LIN {X 0,Y 485.175,Z 367.436,A -85,B 0,C 180,E1 -14967.515,E2 -14967.515} C_VEL
LIN {X 0,Y 481.422,Z 350.009,A -85,B 0,C 180,E1 -14969.767,E2 -14969.767} C_VEL
LIN {X 0,Y 478.767,Z 338.408,A -85,B 0,C 180,E1 -14971.29,E2 -14971.29} C_VEL
LIN {X 0,Y 478.759,Z 338.404,A -85,B 0,C 180,E1 -14973.777,E2 -14973.777} C_VEL
LIN {X 0,Y 478.742,Z 338.407,A -85,B 0,C 180,E1 -14976.861,E2 -14976.861} C_VEL
LIN {X 0,Y 478.759,Z 338.402,A -85,B 0,C 180,E1 -14980.072,E2 -14980.072} C_VEL
LIN {X 0,Y 478.752,Z 338.406,A -85,B 0,C 180,E1 -14983.444,E2 -14983.444} C_VEL
LIN {X 0,Y 478.752,Z 338.406,A -85,B 0,C 180,E1 -14986.556,E2 -14986.556} C_VEL
LIN {X 0,Y 478.766,Z 338.401,A -85,B 0,C 180,E1 -14989.93,E2 -14989.93} C_VEL
LIN {X 0,Y 478.755,Z 338.403,A -85,B 0,C 180,E1 -14993.58,E2 -14993.58} C_VEL
LIN {X 0,Y 478.758,Z 338.409,A -85,B 0,C 180,E1 -14996.506,E2 -14996.506} C_VEL
LIN {X 0,Y 478.73,Z 338.406,A -85,B 0,C 180,E1 -14999.684,E2 -14999.684} C_VEL
LIN {X 0,Y 478.774,Z 338.404,A -85,B 0,C 180,E1 -15002.085,E2 -15002.085} C_VEL
LIN {X 0,Y 478.749,Z 338.404,A -85,B 0,C 180,E1 -15005.109,E2 -15005.109} C_VEL
LIN {X 0,Y 478.778,Z 338.404,A -85,B 0,C 180,E1 -15008.547,E2 -15008.547} C_VEL
LIN {X 0,Y 478.822,Z 338.4,A -85,B 0,C 180,E1 -15011.964,E2 -15011.964} C_VEL
LIN {X 0,Y 478.833,Z 338.4,A -85,B 0,C 180,E1 -15015.708,E2 -15015.708} C_VEL
LIN {X 0,Y 486.096,Z 358.59,A -85,B 0,C 180,E1 -15016.306,E2 -15016.306} C_VEL
LIN {X 0,Y 485.152,Z 454.452,A -85,B 0,C 180,E1 -15017.731,E2 -15017.731} C_VEL
LIN {X 0,Y 485.026,Z 469.135,A -85,B 0,C 180,E1 -15018.072,E2 -15018.072} C_VEL
LIN {X 0,Y 484.751,Z 482.42,A -85,B 0,C 180,E1 -15018.54,E2 -15018.54} C_VEL
LIN {X 0,Y 484.218,Z 495.503,A -85,B 0,C 180,E1 -15019.161,E2 -15019.161} C_VEL
LIN {X 0,Y 483.576,Z 508.953,A -85,B 0,C 180,E1 -15019.99,E2 -15019.99} C_VEL
LIN {X 0,Y 482.964,Z 520.946,A -85,B 0,C 180,E1 -15020.925,E2 -15020.925} C_VEL
LIN {X 0,Y 482.227,Z 530.859,A -85,B 0,C 180,E1 -15021.858,E2 -15021.858} C_VEL
LIN {X 0,Y 481.457,Z 540.12,A -85,B 0,C 180,E1 -15022.897,E2 -15022.897} C_VEL
LIN {X 0,Y 480.63,Z 549.438,A -85,B 0,C 180,E1 -15024.145,E2 -15024.145} C_VEL
LIN {X 0,Y 480.029,Z 557.328,A -85,B 0,C 180,E1 -15025.429,E2 -15025.429} C_VEL
LIN {X 0,Y 479.027,Z 560.589,A -85,B 0,C 180,E1 -15026.007,E2 -15026.007} C_VEL
LIN {X 0,Y 475.742,Z 565.626,A -85,B 0,C 180,E1 -15026.954,E2 -15026.954} C_VEL
LIN {X 0,Y 472.545,Z 570.095,A -85,B 0,C 180,E1 -15027.951,E2 -15027.951} C_VEL
LIN {X 0,Y 471.694,Z 572.465,A -85,B 0,C 180,E1 -15028.599,E2 -15028.599} C_VEL
LIN {X 0,Y 471.381,Z 576.642,A -85,B 0,C 180,E1 -15030,E2 -15030} C_VEL
LIN {X 0,Y 471.202,Z 580.325,A -85,B 0,C 180,E1 -15031.704,E2 -15031.704} C_VEL
LIN {X 0,Y 471.107,Z 582.654,A -85,B 0,C 180,E1 -15033.41,E2 -15033.41} C_VEL
LIN {X 0,Y 471.112,Z 583.684,A -85,B 0,C 180,E1 -15035.118,E2 -15035.118} C_VEL
LIN {X 0,Y 471.242,Z 583.424,A -85,B 0,C 180,E1 -15036.829,E2 -15036.829} C_VEL
LIN {X 0,Y 471.499,Z 581.866,A -85,B 0,C 180,E1 -15038.543,E2 -15038.543} C_VEL
LIN {X 0,Y 471.86,Z 578.968,A -85,B 0,C 180,E1 -15040.261,E2 -15040.261} C_VEL
LIN {X 0,Y 472.534,Z 574.619,A -85,B 0,C 180,E1 -15041.977,E2 -15041.977} C_VEL
LIN {X 0,Y 473.094,Z 570.29,A -85,B 0,C 180,E1 -15043.267,E2 -15043.267} C_VEL
LIN {X 0,Y 473.782,Z 564.997,A -85,B 0,C 180,E1 -15044.556,E2 -15044.556} C_VEL
LIN {X 0,Y 474.765,Z 557.377,A -85,B 0,C 180,E1 -15046.059,E2 -15046.059} C_VEL
LIN {X 0,Y 475.683,Z 549.394,A -85,B 0,C 180,E1 -15047.349,E2 -15047.349} C_VEL
LIN {X 0,Y 476.762,Z 539.731,A -85,B 0,C 180,E1 -15048.636,E2 -15048.636} C_VEL
LIN {X 0,Y 477.733,Z 530.02,A -85,B 0,C 180,E1 -15049.708,E2 -15049.708} C_VEL
LIN {X 0,Y 478.639,Z 519.536,A -85,B 0,C 180,E1 -15050.674,E2 -15050.674} C_VEL
LIN {X 0,Y 479.678,Z 506.651,A -85,B 0,C 180,E1 -15051.636,E2 -15051.636} C_VEL
LIN {X 0,Y 480.39,Z 493.952,A -85,B 0,C 180,E1 -15052.391,E2 -15052.391} C_VEL
LIN {X 0,Y 480.884,Z 480.962,A -85,B 0,C 180,E1 -15052.989,E2 -15052.989} C_VEL
LIN {X 0,Y 481.254,Z 467.044,A -85,B 0,C 180,E1 -15053.452,E2 -15053.452} C_VEL
LIN {X 0,Y 481.406,Z 452.358,A -85,B 0,C 180,E1 -15053.757,E2 -15053.757} C_VEL
LIN {X 0,Y 482.688,Z 365.012,A -85,B 0,C 180,E1 -15055.071,E2 -15055.071} C_VEL
LIN {X 0,Y 472.549,Z 341.866,A -85,B 0,C 180,E1 -15055.964,E2 -15055.964} C_VEL
LIN {X 0,Y 471.684,Z 339.29,A -85,B 0,C 180,E1 -15056.066,E2 -15056.066} C_VEL
LIN {X 0,Y 471.685,Z 339.289,A -85,B 0,C 180,E1 -15059.344,E2 -15059.344} C_VEL
LIN {X 0,Y 471.624,Z 339.297,A -85,B 0,C 180,E1 -15062.321,E2 -15062.321} C_VEL
LIN {X 0,Y 471.636,Z 339.292,A -85,B 0,C 180,E1 -15065.395,E2 -15065.395} C_VEL
LIN {X 0,Y 471.628,Z 339.296,A -85,B 0,C 180,E1 -15068.592,E2 -15068.592} C_VEL
LIN {X 0,Y 471.672,Z 339.29,A -85,B 0,C 180,E1 -15070.8,E2 -15070.8} C_VEL
LIN {X 0,Y 471.685,Z 339.287,A -85,B 0,C 180,E1 -15074.263,E2 -15074.263} C_VEL
LIN {X 0,Y 471.681,Z 339.286,A -85,B 0,C 180,E1 -15076.913,E2 -15076.913} C_VEL
LIN {X 0,Y 471.673,Z 339.286,A -85,B 0,C 180,E1 -15079.233,E2 -15079.233} C_VEL
LIN {X 0,Y 471.624,Z 339.268,A -85,B 0,C 180,E1 -15082.488,E2 -15082.488} C_VEL
LIN {X 0,Y 471.659,Z 339.279,A -85,B 0,C 180,E1 -15085.644,E2 -15085.644} C_VEL
LIN {X 0,Y 471.649,Z 339.282,A -85,B 0,C 180,E1 -15088.682,E2 -15088.682} C_VEL
LIN {X 0,Y 471.696,Z 339.286,A -85,B 0,C 180,E1 -15091.628,E2 -15091.628} C_VEL
LIN {X 0,Y 471.698,Z 339.277,A -85,B 0,C 180,E1 -15094.934,E2 -15094.934} C_VEL
LIN {X 0,Y 471.653,Z 339.283,A -85,B 0,C 180,E1 -15098.206,E2 -15098.206} C_VEL
LIN {X 0,Y 471.723,Z 339.286,A -85,B 0,C 180,E1 -15100.414,E2 -15100.414} C_VEL
LIN {X 0,Y 477.254,Z 358.133,A -85,B 0,C 180,E1 -15100.948,E2 -15100.948} C_VEL
LIN {X 0,Y 475.404,Z 458.142,A -85,B 0,C 180,E1 -15102.884,E2 -15102.884} C_VEL
LIN {X 0,Y 475.207,Z 473.733,A -85,B 0,C 180,E1 -15103.372,E2 -15103.372} C_VEL
LIN {X 0,Y 474.822,Z 488.087,A -85,B 0,C 180,E1 -15103.998,E2 -15103.998} C_VEL
LIN {X 0,Y 474.305,Z 502.141,A -85,B 0,C 180,E1 -15104.803,E2 -15104.803} C_VEL
LIN {X 0,Y 473.779,Z 515.566,A -85,B 0,C 180,E1 -15105.771,E2 -15105.771} C_VEL
LIN {X 0,Y 473.158,Z 527.661,A -85,B 0,C 180,E1 -15106.844,E2 -15106.844} C_VEL
LIN {X 0,Y 472.756,Z 538.588,A -85,B 0,C 180,E1 -15108.028,E2 -15108.028} C_VEL
LIN {X 0,Y 472.269,Z 548.47,A -85,B 0,C 180,E1 -15109.316,E2 -15109.316} C_VEL
LIN {X 0,Y 471.798,Z 556.687,A -85,B 0,C 180,E1 -15110.601,E2 -15110.601} C_VEL
LIN {X 0,Y 471.436,Z 564.576,A -85,B 0,C 180,E1 -15112.1,E2 -15112.1} C_VEL
LIN {X 0,Y 471.186,Z 570.862,A -85,B 0,C 180,E1 -15113.598,E2 -15113.598} C_VEL
LIN {X 0,Y 471.065,Z 575.618,A -85,B 0,C 180,E1 -15115.04,E2 -15115.04} C_VEL
LIN {X 0,Y 471.062,Z 579.426,A -85,B 0,C 180,E1 -15116.59,E2 -15116.59} C_VEL
LIN {X 0,Y 471.048,Z 582.191,A -85,B 0,C 180,E1 -15118.296,E2 -15118.296} C_VEL
LIN {X 0,Y 471.138,Z 583.53,A -85,B 0,C 180,E1 -15120,E2 -15120} C_VEL
LIN {X 0,Y 471.354,Z 583.455,A -85,B 0,C 180,E1 -15121.703,E2 -15121.703} C_VEL
LIN {X 0,Y 471.885,Z 581.884,A -85,B 0,C 180,E1 -15123.404,E2 -15123.404} C_VEL
LIN {X 0,Y 472.565,Z 578.84,A -85,B 0,C 180,E1 -15125.102,E2 -15125.102} C_VEL
LIN {X 0,Y 473.152,Z 574.316,A -85,B 0,C 180,E1 -15126.801,E2 -15126.801} C_VEL
LIN {X 0,Y 474.083,Z 569.426,A -85,B 0,C 180,E1 -15128.145,E2 -15128.145} C_VEL
LIN {X 0,Y 475.187,Z 562.024,A -85,B 0,C 180,E1 -15129.759,E2 -15129.759} C_VEL
LIN {X 0,Y 476.091,Z 554.81,A -85,B 0,C 180,E1 -15131.026,E2 -15131.026} C_VEL
LIN {X 0,Y 477.182,Z 546.051,A -85,B 0,C 180,E1 -15132.289,E2 -15132.289} C_VEL
LIN {X 0,Y 478.244,Z 535.494,A -85,B 0,C 180,E1 -15133.552,E2 -15133.552} C_VEL
LIN {X 0,Y 479.504,Z 523.618,A -85,B 0,C 180,E1 -15134.703,E2 -15134.703} C_VEL
LIN {X 0,Y 480.668,Z 511.003,A -85,B 0,C 180,E1 -15135.681,E2 -15135.681} C_VEL
LIN {X 0,Y 481.659,Z 497.123,A -85,B 0,C 180,E1 -15136.55,E2 -15136.55} C_VEL
LIN {X 0,Y 482.27,Z 483.595,A -85,B 0,C 180,E1 -15137.213,E2 -15137.213} C_VEL
LIN {X 0,Y 482.778,Z 468.86,A -85,B 0,C 180,E1 -15137.739,E2 -15137.739} C_VEL
LIN {X 0,Y 483.214,Z 450.578,A -85,B 0,C 180,E1 -15138.186,E2 -15138.186} C_VEL
LIN {X 0,Y 486.455,Z 378.243,A -85,B 0,C 180,E1 -15139.782,E2 -15139.782} C_VEL
LIN {X 0,Y 486.873,Z 368.471,A -85,B 0,C 180,E1 -15140.011,E2 -15140.011} C_VEL
LIN {X 0,Y 480.186,Z 354.884,A -85,B 0,C 180,E1 -15140.946,E2 -15140.946} C_VEL
LIN {X 0,Y 475.319,Z 346.362,A -85,B 0,C 180,E1 -15141.636,E2 -15141.636} C_VEL
LIN {X 0,Y 473.366,Z 343.01,A -85,B 0,C 180,E1 -15141.922,E2 -15141.922} C_VEL
LIN {X 0,Y 471.939,Z 340.35,A -85,B 0,C 180,E1 -15142.149,E2 -15142.149} C_VEL
LIN {X 0,Y 471.737,Z 339.286,A -85,B 0,C 180,E1 -15142.215,E2 -15142.215} C_VEL
LIN {X 0,Y 471.713,Z 339.288,A -85,B 0,C 180,E1 -15145.507,E2 -15145.507} C_VEL
LIN {X 0,Y 471.71,Z 339.286,A -85,B 0,C 180,E1 -15148.37,E2 -15148.37} C_VEL
LIN {X 0,Y 471.69,Z 339.289,A -85,B 0,C 180,E1 -15151.315,E2 -15151.315} C_VEL
LIN {X 0,Y 471.7,Z 339.282,A -85,B 0,C 180,E1 -15154.352,E2 -15154.352} C_VEL
LIN {X 0,Y 471.67,Z 339.284,A -85,B 0,C 180,E1 -15157.507,E2 -15157.507} C_VEL
LIN {X 0,Y 471.682,Z 339.283,A -85,B 0,C 180,E1 -15159.683,E2 -15159.683} C_VEL
LIN {X 0,Y 471.679,Z 339.285,A -85,B 0,C 180,E1 -15163.086,E2 -15163.086} C_VEL
LIN {X 0,Y 471.686,Z 339.283,A -85,B 0,C 180,E1 -15165.738,E2 -15165.738} C_VEL
LIN {X 0,Y 471.67,Z 339.289,A -85,B 0,C 180,E1 -15169.232,E2 -15169.232} C_VEL
LIN {X 0,Y 471.622,Z 339.298,A -85,B 0,C 180,E1 -15172.488,E2 -15172.488} C_VEL
LIN {X 0,Y 471.629,Z 339.285,A -85,B 0,C 180,E1 -15175.642,E2 -15175.642} C_VEL
LIN {X 0,Y 471.674,Z 339.381,A -85,B 0,C 180,E1 -15177.525,E2 -15177.525} C_VEL
LIN {X 0,Y 475.594,Z 355.323,A -85,B 0,C 180,E1 -15180.107,E2 -15180.107} C_VEL
LIN {X 0,Y 478.251,Z 367.913,A -85,B 0,C 180,E1 -15182.052,E2 -15182.052} C_VEL
LIN {X 0,Y 478.074,Z 372.934,A -85,B 0,C 180,E1 -15182.751,E2 -15182.751} C_VEL
LIN {X 0,Y 475.774,Z 399.746,A -85,B 0,C 180,E1 -15186.378,E2 -15186.378} C_VEL
LIN {X 0,Y 475.192,Z 407.187,A -85,B 0,C 180,E1 -15187.379,E2 -15187.379} C_VEL
LIN {X 0,Y 478.527,Z 428.614,A -85,B 0,C 180,E1 -15188.267,E2 -15188.267} C_VEL
LIN {X 0,Y 480.639,Z 445.485,A -85,B 0,C 180,E1 -15188.882,E2 -15188.882} C_VEL
LIN {X 0,Y 482.569,Z 472.55,A -85,B 0,C 180,E1 -15189.724,E2 -15189.724} C_VEL
LIN {X 0,Y 480.102,Z 533.094,A -85,B 0,C 180,E1 -15191.03,E2 -15191.03} C_VEL
LIN {X 0,Y 479.615,Z 559.637,A -85,B 0,C 180,E1 -15191.452,E2 -15191.452} C_VEL
LIN {X 0,Y 478.87,Z 573.984,A -85,B 0,C 180,E1 -15191.836,E2 -15191.836} C_VEL
LIN {X 0,Y 477.735,Z 588.728,A -85,B 0,C 180,E1 -15192.415,E2 -15192.415} C_VEL
LIN {X 0,Y 476.54,Z 602.089,A -85,B 0,C 180,E1 -15193.124,E2 -15193.124} C_VEL
LIN {X 0,Y 475.343,Z 614.425,A -85,B 0,C 180,E1 -15193.961,E2 -15193.961} C_VEL
LIN {X 0,Y 474.022,Z 626.919,A -85,B 0,C 180,E1 -15195.013,E2 -15195.013} C_VEL
LIN {X 0,Y 472.917,Z 637.198,A -85,B 0,C 180,E1 -15196.073,E2 -15196.073} C_VEL
LIN {X 0,Y 472.057,Z 647.255,A -85,B 0,C 180,E1 -15197.303,E2 -15197.303} C_VEL
LIN {X 0,Y 471.418,Z 658.908,A -85,B 0,C 180,E1 -15198.472,E2 -15198.472} C_VEL
LIN {X 0,Y 470.946,Z 669.094,A -85,B 0,C 180,E1 -15199.719,E2 -15199.719} C_VEL
LIN {X 0,Y 470.512,Z 677.788,A -85,B 0,C 180,E1 -15201.007,E2 -15201.007} C_VEL
LIN {X 0,Y 470.174,Z 686.056,A -85,B 0,C 180,E1 -15202.51,E2 -15202.51} C_VEL
LIN {X 0,Y 470.009,Z 692.665,A -85,B 0,C 180,E1 -15204.012,E2 -15204.012} C_VEL
LIN {X 0,Y 469.925,Z 697.153,A -85,B 0,C 180,E1 -15205.297,E2 -15205.297} C_VEL
LIN {X 0,Y 469.843,Z 700.68,A -85,B 0,C 180,E1 -15206.581,E2 -15206.581} C_VEL
LIN {X 0,Y 469.856,Z 702.494,A -85,B 0,C 180,E1 -15207.437,E2 -15207.437} C_VEL
LIN {X 0,Y 469.847,Z 704.973,A -85,B 0,C 180,E1 -15209.146,E2 -15209.146} C_VEL
LIN {X 0,Y 469.83,Z 705.968,A -85,B 0,C 180,E1 -15210.854,E2 -15210.854} C_VEL
LIN {X 0,Y 469.856,Z 705.494,A -85,B 0,C 180,E1 -15212.563,E2 -15212.563} C_VEL
LIN {X 0,Y 469.942,Z 703.555,A -85,B 0,C 180,E1 -15214.274,E2 -15214.274} C_VEL
LIN {X 0,Y 470.23,Z 700.082,A -85,B 0,C 180,E1 -15215.985,E2 -15215.985} C_VEL
LIN {X 0,Y 470.588,Z 695.019,A -85,B 0,C 180,E1 -15217.698,E2 -15217.698} C_VEL
LIN {X 0,Y 471.087,Z 690.095,A -85,B 0,C 180,E1 -15218.982,E2 -15218.982} C_VEL
LIN {X 0,Y 471.897,Z 682.967,A -85,B 0,C 180,E1 -15220.476,E2 -15220.476} C_VEL
LIN {X 0,Y 472.829,Z 674.129,A -85,B 0,C 180,E1 -15221.97,E2 -15221.97} C_VEL
LIN {X 0,Y 473.827,Z 664.913,A -85,B 0,C 180,E1 -15223.246,E2 -15223.246} C_VEL
LIN {X 0,Y 475.122,Z 653.768,A -85,B 0,C 180,E1 -15224.514,E2 -15224.514} C_VEL
LIN {X 0,Y 476.226,Z 642.496,A -85,B 0,C 180,E1 -15225.571,E2 -15225.571} C_VEL
LIN {X 0,Y 477.639,Z 628.699,A -85,B 0,C 180,E1 -15226.616,E2 -15226.616} C_VEL
LIN {X 0,Y 478.836,Z 614.862,A -85,B 0,C 180,E1 -15227.45,E2 -15227.45} C_VEL
LIN {X 0,Y 479.94,Z 600.174,A -85,B 0,C 180,E1 -15228.121,E2 -15228.121} C_VEL
LIN {X 0,Y 480.96,Z 584.717,A -85,B 0,C 180,E1 -15228.631,E2 -15228.631} C_VEL
LIN {X 0,Y 485.642,Z 483.73,A -85,B 0,C 180,E1 -15230.914,E2 -15230.914} C_VEL
LIN {X 0,Y 486.051,Z 471.893,A -85,B 0,C 180,E1 -15231.207,E2 -15231.207} C_VEL
LIN {X 0,Y 485.065,Z 454.594,A -85,B 0,C 180,E1 -15231.77,E2 -15231.77} C_VEL
LIN {X 0,Y 482.938,Z 436.376,A -85,B 0,C 180,E1 -15232.478,E2 -15232.478} C_VEL
LIN {X 0,Y 481.981,Z 418.453,A -85,B 0,C 180,E1 -15233.573,E2 -15233.573} C_VEL
LIN {X 0,Y 480.737,Z 398.185,A -85,B 0,C 180,E1 -15234.995,E2 -15234.995} C_VEL
LIN {X 0,Y 479.656,Z 383.288,A -85,B 0,C 180,E1 -15236.196,E2 -15236.196} C_VEL
LIN {X 0,Y 479.315,Z 374.608,A -85,B 0,C 180,E1 -15236.948,E2 -15236.948} C_VEL
LIN {X 0,Y 478.81,Z 365.879,A -85,B 0,C 180,E1 -15237.783,E2 -15237.783} C_VEL
LIN {X 0,Y 476.954,Z 356.575,A -85,B 0,C 180,E1 -15238.988,E2 -15238.988} C_VEL
LIN {X 0,Y 474.733,Z 345.236,A -85,B 0,C 180,E1 -15240.717,E2 -15240.717} C_VEL
LIN {X 0,Y 474.115,Z 343.792,A -85,B 0,C 180,E1 -15241.032,E2 -15241.032} C_VEL
LIN {X 0,Y 472.071,Z 340.988,A -85,B 0,C 180,E1 -15241.91,E2 -15241.91} C_VEL
LIN {X 0,Y 471.613,Z 339.294,A -85,B 0,C 180,E1 -15242.322,E2 -15242.322} C_VEL
LIN {X 0,Y 471.624,Z 339.292,A -85,B 0,C 180,E1 -15245.396,E2 -15245.396} C_VEL
LIN {X 0,Y 471.622,Z 339.295,A -85,B 0,C 180,E1 -15248.592,E2 -15248.592} C_VEL
LIN {X 0,Y 471.667,Z 339.288,A -85,B 0,C 180,E1 -15250.8,E2 -15250.8} C_VEL
LIN {X 0,Y 471.681,Z 339.291,A -85,B 0,C 180,E1 -15254.263,E2 -15254.263} C_VEL
LIN {X 0,Y 471.664,Z 339.287,A -85,B 0,C 180,E1 -15256.912,E2 -15256.912} C_VEL
LIN {X 0,Y 471.668,Z 339.29,A -85,B 0,C 180,E1 -15259.233,E2 -15259.233} C_VEL
LIN {X 0,Y 471.648,Z 339.291,A -85,B 0,C 180,E1 -15260.47,E2 -15260.47} C_VEL
LIN {X 0,Y 472.464,Z 341.824,A -85,B 0,C 180,E1 -15261.214,E2 -15261.214} C_VEL
LIN {X 0,Y 474.12,Z 344.845,A -85,B 0,C 180,E1 -15262.195,E2 -15262.195} C_VEL
LIN {X 0,Y 477.879,Z 353.112,A -85,B 0,C 180,E1 -15264.437,E2 -15264.437} C_VEL
LIN {X 0,Y 481.184,Z 361.878,A -85,B 0,C 180,E1 -15266.416,E2 -15266.416} C_VEL
LIN {X 0,Y 483.952,Z 370.881,A -85,B 0,C 180,E1 -15268.196,E2 -15268.196} C_VEL
LIN {X 0,Y 486.231,Z 379.99,A -85,B 0,C 180,E1 -15269.807,E2 -15269.807} C_VEL
LIN {X 0,Y 486.938,Z 383.965,A -85,B 0,C 180,E1 -15270.459,E2 -15270.459} C_VEL
LIN {X 0,Y 486.785,Z 387.543,A -85,B 0,C 180,E1 -15270.946,E2 -15270.946} C_VEL
LIN {X 0,Y 484.134,Z 412.267,A -85,B 0,C 180,E1 -15274.03,E2 -15274.03} C_VEL
LIN {X 0,Y 481.588,Z 440.052,A -85,B 0,C 180,E1 -15277.429,E2 -15277.429} C_VEL
LIN {X 0,Y 485.077,Z 458.784,A -85,B 0,C 180,E1 -15278.258,E2 -15278.258} C_VEL
LIN {X 0,Y 486.657,Z 471.979,A -85,B 0,C 180,E1 -15278.747,E2 -15278.747} C_VEL
LIN {X 0,Y 482.69,Z 556.46,A -85,B 0,C 180,E1 -15280.645,E2 -15280.645} C_VEL
LIN {X 0,Y 481.474,Z 583.391,A -85,B 0,C 180,E1 -15281.26,E2 -15281.26} C_VEL
LIN {X 0,Y 480.568,Z 596.124,A -85,B 0,C 180,E1 -15281.683,E2 -15281.683} C_VEL
LIN {X 0,Y 479.389,Z 610.913,A -85,B 0,C 180,E1 -15282.351,E2 -15282.351} C_VEL
LIN {X 0,Y 478.219,Z 624.997,A -85,B 0,C 180,E1 -15283.185,E2 -15283.185} C_VEL
LIN {X 0,Y 476.917,Z 637.696,A -85,B 0,C 180,E1 -15284.125,E2 -15284.125} C_VEL
LIN {X 0,Y 475.637,Z 649.296,A -85,B 0,C 180,E1 -15285.175,E2 -15285.175} C_VEL
LIN {X 0,Y 474.467,Z 659.905,A -85,B 0,C 180,E1 -15286.338,E2 -15286.338} C_VEL
LIN {X 0,Y 473.279,Z 669.716,A -85,B 0,C 180,E1 -15287.631,E2 -15287.631} C_VEL
LIN {X 0,Y 472.382,Z 678.846,A -85,B 0,C 180,E1 -15289.102,E2 -15289.102} C_VEL
LIN {X 0,Y 471.36,Z 686.341,A -85,B 0,C 180,E1 -15290.592,E2 -15290.592} C_VEL
LIN {X 0,Y 470.839,Z 691.557,A -85,B 0,C 180,E1 -15291.876,E2 -15291.876} C_VEL
LIN {X 0,Y 470.435,Z 695.757,A -85,B 0,C 180,E1 -15293.159,E2 -15293.159} C_VEL
LIN {X 0,Y 470.034,Z 699.981,A -85,B 0,C 180,E1 -15294.87,E2 -15294.87} C_VEL
LIN {X 0,Y 469.847,Z 702.671,A -85,B 0,C 180,E1 -15296.582,E2 -15296.582} C_VEL
LIN {X 0,Y 469.765,Z 703.876,A -85,B 0,C 180,E1 -15298.291,E2 -15298.291} C_VEL
LIN {X 0,Y 469.76,Z 703.636,A -85,B 0,C 180,E1 -15300,E2 -15300} C_VEL
LIN {X 0,Y 469.76,Z 701.944,A -85,B 0,C 180,E1 -15301.709,E2 -15301.709} C_VEL
LIN {X 0,Y 469.809,Z 698.766,A -85,B 0,C 180,E1 -15303.419,E2 -15303.419} C_VEL
LIN {X 0,Y 469.863,Z 695.314,A -85,B 0,C 180,E1 -15304.703,E2 -15304.703} C_VEL
LIN {X 0,Y 469.993,Z 690.848,A -85,B 0,C 180,E1 -15306.008,E2 -15306.008} C_VEL
LIN {X 0,Y 470.256,Z 684.46,A -85,B 0,C 180,E1 -15307.489,E2 -15307.489} C_VEL
LIN {X 0,Y 470.579,Z 676.37,A -85,B 0,C 180,E1 -15308.992,E2 -15308.992} C_VEL
LIN {X 0,Y 471.047,Z 667.898,A -85,B 0,C 180,E1 -15310.279,E2 -15310.279} C_VEL
LIN {X 0,Y 471.568,Z 658.05,A -85,B 0,C 180,E1 -15311.524,E2 -15311.524} C_VEL
LIN {X 0,Y 472.122,Z 647.404,A -85,B 0,C 180,E1 -15312.641,E2 -15312.641} C_VEL
LIN {X 0,Y 472.792,Z 634.963,A -85,B 0,C 180,E1 -15313.712,E2 -15313.712} C_VEL
LIN {X 0,Y 473.52,Z 622.844,A -85,B 0,C 180,E1 -15314.565,E2 -15314.565} C_VEL
LIN {X 0,Y 474.22,Z 608.634,A -85,B 0,C 180,E1 -15315.364,E2 -15315.364} C_VEL
LIN {X 0,Y 474.712,Z 594.201,A -85,B 0,C 180,E1 -15315.979,E2 -15315.979} C_VEL
LIN {X 0,Y 475.181,Z 579.664,A -85,B 0,C 180,E1 -15316.417,E2 -15316.417} C_VEL
LIN {X 0,Y 477.528,Z 466.879,A -85,B 0,C 180,E1 -15318.632,E2 -15318.632} C_VEL
LIN {X 0,Y 474.708,Z 439.522,A -85,B 0,C 180,E1 -15319.275,E2 -15319.275} C_VEL
LIN {X 0,Y 476.23,Z 408.418,A -85,B 0,C 180,E1 -15322.94,E2 -15322.94} C_VEL
LIN {X 0,Y 477.57,Z 383.579,A -85,B 0,C 180,E1 -15325.871,E2 -15325.871} C_VEL
LIN {X 0,Y 478.296,Z 370.046,A -85,B 0,C 180,E1 -15327.472,E2 -15327.472} C_VEL
LIN {X 0,Y 477.248,Z 363.687,A -85,B 0,C 180,E1 -15328.285,E2 -15328.285} C_VEL
LIN {X 0,Y 472.51,Z 342.754,A -85,B 0,C 180,E1 -15331.04,E2 -15331.04} C_VEL
LIN {X 0,Y 471.716,Z 339.286,A -85,B 0,C 180,E1 -15331.5,E2 -15331.5} C_VEL
LIN {X 0,Y 471.701,Z 339.281,A -85,B 0,C 180,E1 -15334.352,E2 -15334.352} C_VEL
LIN {X 0,Y 471.671,Z 339.289,A -85,B 0,C 180,E1 -15337.508,E2 -15337.508} C_VEL
LIN {X 0,Y 471.721,Z 339.28,A -85,B 0,C 180,E1 -15339.68,E2 -15339.68} C_VEL
LIN {X 0,Y 471.697,Z 339.286,A -85,B 0,C 180,E1 -15343.312,E2 -15343.312} C_VEL
LIN {X 0,Y 471.707,Z 339.281,A -85,B 0,C 180,E1 -15345.74,E2 -15345.74} C_VEL
LIN {X 0,Y 471.707,Z 339.284,A -85,B 0,C 180,E1 -15349.228,E2 -15349.228} C_VEL
LIN {X 0,Y 471.663,Z 339.286,A -85,B 0,C 180,E1 -15351.914,E2 -15351.914} C_VEL
LIN {X 0,Y 471.699,Z 339.288,A -85,B 0,C 180,E1 -15354.758,E2 -15354.758} C_VEL
LIN {X 0,Y 471.694,Z 339.283,A -85,B 0,C 180,E1 -15357.826,E2 -15357.826} C_VEL
LIN {X 0,Y 471.69,Z 339.288,A -85,B 0,C 180,E1 -15360.657,E2 -15360.657} C_VEL
LIN {X 0,Y 471.693,Z 339.282,A -85,B 0,C 180,E1 -15363.545,E2 -15363.545} C_VEL
LIN {X 0,Y 471.68,Z 339.291,A -85,B 0,C 180,E1 -15366.362,E2 -15366.362} C_VEL
LIN {X 0,Y 471.758,Z 339.274,A -85,B 0,C 180,E1 -15369.293,E2 -15369.293} C_VEL
LIN {X 0,Y 471.727,Z 339.279,A -85,B 0,C 180,E1 -15372.724,E2 -15372.724} C_VEL
LIN {X 0,Y 471.783,Z 339.31,A -85,B 0,C 180,E1 -15375.451,E2 -15375.451} C_VEL
LIN {X 0,Y 479.432,Z 360.627,A -85,B 0,C 180,E1 -15376.085,E2 -15376.085} C_VEL
LIN {X 0,Y 478.337,Z 454.876,A -85,B 0,C 180,E1 -15377.5,E2 -15377.5} C_VEL
LIN {X 0,Y 478.205,Z 469.692,A -85,B 0,C 180,E1 -15377.845,E2 -15377.845} C_VEL
LIN {X 0,Y 477.936,Z 483.032,A -85,B 0,C 180,E1 -15378.321,E2 -15378.321} C_VEL
LIN {X 0,Y 477.417,Z 495.178,A -85,B 0,C 180,E1 -15378.898,E2 -15378.898} C_VEL
LIN {X 0,Y 476.824,Z 507.302,A -85,B 0,C 180,E1 -15379.633,E2 -15379.633} C_VEL
LIN {X 0,Y 476.228,Z 519.045,A -85,B 0,C 180,E1 -15380.522,E2 -15380.522} C_VEL
LIN {X 0,Y 475.475,Z 529.982,A -85,B 0,C 180,E1 -15381.529,E2 -15381.529} C_VEL
LIN {X 0,Y 474.656,Z 539.52,A -85,B 0,C 180,E1 -15382.581,E2 -15382.581} C_VEL
LIN {X 0,Y 473.743,Z 549.071,A -85,B 0,C 180,E1 -15383.847,E2 -15383.847} C_VEL
LIN {X 0,Y 473.162,Z 556.969,A -85,B 0,C 180,E1 -15385.117,E2 -15385.117} C_VEL
LIN {X 0,Y 472.38,Z 564.575,A -85,B 0,C 180,E1 -15386.6,E2 -15386.6} C_VEL
LIN {X 0,Y 471.964,Z 569.878,A -85,B 0,C 180,E1 -15387.874,E2 -15387.874} C_VEL
LIN {X 0,Y 471.694,Z 572.465,A -85,B 0,C 180,E1 -15388.599,E2 -15388.599} C_VEL
LIN {X 0,Y 470.861,Z 574.662,A -85,B 0,C 180,E1 -15389.26,E2 -15389.26} C_VEL
LIN {X 0,Y 467.796,Z 577.914,A -85,B 0,C 180,E1 -15390.342,E2 -15390.342} C_VEL
LIN {X 0,Y 465.29,Z 580.129,A -85,B 0,C 180,E1 -15391.229,E2 -15391.229} C_VEL
LIN {X 0,Y 464.229,Z 581.485,A -85,B 0,C 180,E1 -15391.927,E2 -15391.927} C_VEL
LIN {X 0,Y 464.148,Z 581.826,A -85,B 0,C 180,E1 -15392.166,E2 -15392.166} C_VEL
LIN {X 0,Y 464.04,Z 583.466,A -85,B 0,C 180,E1 -15393.462,E2 -15393.462} C_VEL
LIN {X 0,Y 464.071,Z 584.46,A -85,B 0,C 180,E1 -15395.196,E2 -15395.196} C_VEL
LIN {X 0,Y 464.215,Z 584.167,A -85,B 0,C 180,E1 -15396.933,E2 -15396.933} C_VEL
LIN {X 0,Y 464.465,Z 582.577,A -85,B 0,C 180,E1 -15398.674,E2 -15398.674} C_VEL
LIN {X 0,Y 464.886,Z 579.64,A -85,B 0,C 180,E1 -15400.417,E2 -15400.417} C_VEL
LIN {X 0,Y 465.586,Z 575.254,A -85,B 0,C 180,E1 -15402.159,E2 -15402.159} C_VEL
LIN {X 0,Y 466.168,Z 570.886,A -85,B 0,C 180,E1 -15403.468,E2 -15403.468} C_VEL
LIN {X 0,Y 466.904,Z 565.549,A -85,B 0,C 180,E1 -15404.776,E2 -15404.776} C_VEL
LIN {X 0,Y 467.925,Z 557.881,A -85,B 0,C 180,E1 -15406.301,E2 -15406.301} C_VEL
LIN {X 0,Y 468.889,Z 549.843,A -85,B 0,C 180,E1 -15407.608,E2 -15407.608} C_VEL
LIN {X 0,Y 470.013,Z 540.115,A -85,B 0,C 180,E1 -15408.913,E2 -15408.913} C_VEL
LIN {X 0,Y 471.035,Z 530.326,A -85,B 0,C 180,E1 -15410,E2 -15410} C_VEL
LIN {X 0,Y 472,Z 519.744,A -85,B 0,C 180,E1 -15410.978,E2 -15410.978} C_VEL
LIN {X 0,Y 472.932,Z 508.31,A -85,B 0,C 180,E1 -15411.847,E2 -15411.847} C_VEL
LIN {X 0,Y 473.715,Z 495.842,A -85,B 0,C 180,E1 -15412.609,E2 -15412.609} C_VEL
LIN {X 0,Y 474.214,Z 483.203,A -85,B 0,C 180,E1 -15413.216,E2 -15413.216} C_VEL
LIN {X 0,Y 474.627,Z 468.884,A -85,B 0,C 180,E1 -15413.716,E2 -15413.716} C_VEL
LIN {X 0,Y 474.805,Z 455.104,A -85,B 0,C 180,E1 -15414.024,E2 -15414.024} C_VEL
LIN {X 0,Y 476.177,Z 366.885,A -85,B 0,C 180,E1 -15415.37,E2 -15415.37} C_VEL
LIN {X 0,Y 465.674,Z 343.092,A -85,B 0,C 180,E1 -15416.315,E2 -15416.315} C_VEL
LIN {X 0,Y 464.624,Z 340.17,A -85,B 0,C 180,E1 -15416.423,E2 -15416.423} C_VEL
LIN {X 0,Y 464.668,Z 340.164,A -85,B 0,C 180,E1 -15419.037,E2 -15419.037} C_VEL
LIN {X 0,Y 464.597,Z 340.172,A -85,B 0,C 180,E1 -15422.405,E2 -15422.405} C_VEL
LIN {X 0,Y 464.583,Z 340.171,A -85,B 0,C 180,E1 -15425.496,E2 -15425.496} C_VEL
LIN {X 0,Y 464.585,Z 340.176,A -85,B 0,C 180,E1 -15428.372,E2 -15428.372} C_VEL
LIN {X 0,Y 464.622,Z 340.169,A -85,B 0,C 180,E1 -15431.554,E2 -15431.554} C_VEL
LIN {X 0,Y 464.671,Z 340.156,A -85,B 0,C 180,E1 -15435.112,E2 -15435.112} C_VEL
LIN {X 0,Y 464.629,Z 340.165,A -85,B 0,C 180,E1 -15438.446,E2 -15438.446} C_VEL
LIN {X 0,Y 464.575,Z 340.155,A -85,B 0,C 180,E1 -15441.818,E2 -15441.818} C_VEL
LIN {X 0,Y 464.621,Z 340.151,A -85,B 0,C 180,E1 -15445.049,E2 -15445.049} C_VEL
LIN {X 0,Y 464.582,Z 340.167,A -85,B 0,C 180,E1 -15448.15,E2 -15448.15} C_VEL
LIN {X 0,Y 464.659,Z 340.158,A -85,B 0,C 180,E1 -15451.159,E2 -15451.159} C_VEL
LIN {X 0,Y 464.648,Z 340.156,A -85,B 0,C 180,E1 -15454.076,E2 -15454.076} C_VEL
LIN {X 0,Y 464.63,Z 340.164,A -85,B 0,C 180,E1 -15456.923,E2 -15456.923} C_VEL
LIN {X 0,Y 464.692,Z 340.163,A -85,B 0,C 180,E1 -15460.243,E2 -15460.243} C_VEL
LIN {X 0,Y 470.238,Z 358.755,A -85,B 0,C 180,E1 -15460.781,E2 -15460.781} C_VEL
LIN {X 0,Y 468.391,Z 458.568,A -85,B 0,C 180,E1 -15462.759,E2 -15462.759} C_VEL
LIN {X 0,Y 468.183,Z 473.722,A -85,B 0,C 180,E1 -15463.237,E2 -15463.237} C_VEL
LIN {X 0,Y 467.817,Z 488.047,A -85,B 0,C 180,E1 -15463.863,E2 -15463.863} C_VEL
LIN {X 0,Y 467.346,Z 500.625,A -85,B 0,C 180,E1 -15464.571,E2 -15464.571} C_VEL
LIN {X 0,Y 466.892,Z 513.081,A -85,B 0,C 180,E1 -15465.446,E2 -15465.446} C_VEL
LIN {X 0,Y 466.269,Z 525.734,A -85,B 0,C 180,E1 -15466.535,E2 -15466.535} C_VEL
LIN {X 0,Y 465.81,Z 536.226,A -85,B 0,C 180,E1 -15467.626,E2 -15467.626} C_VEL
LIN {X 0,Y 465.34,Z 546.718,A -85,B 0,C 180,E1 -15468.935,E2 -15468.935} C_VEL
LIN {X 0,Y 464.871,Z 555.375,A -85,B 0,C 180,E1 -15470.24,E2 -15470.24} C_VEL
LIN {X 0,Y 464.452,Z 563.643,A -85,B 0,C 180,E1 -15471.763,E2 -15471.763} C_VEL
LIN {X 0,Y 464.198,Z 569.45,A -85,B 0,C 180,E1 -15473.066,E2 -15473.066} C_VEL
LIN {X 0,Y 464.031,Z 574.203,A -85,B 0,C 180,E1 -15474.369,E2 -15474.369} C_VEL
LIN {X 0,Y 463.997,Z 577.973,A -85,B 0,C 180,E1 -15475.671,E2 -15475.671} C_VEL
LIN {X 0,Y 464.027,Z 581.62,A -85,B 0,C 180,E1 -15477.404,E2 -15477.404} C_VEL
LIN {X 0,Y 464.023,Z 583.789,A -85,B 0,C 180,E1 -15479.135,E2 -15479.135} C_VEL
LIN {X 0,Y 464.206,Z 584.536,A -85,B 0,C 180,E1 -15480.864,E2 -15480.864} C_VEL
LIN {X 0,Y 464.567,Z 583.856,A -85,B 0,C 180,E1 -15482.592,E2 -15482.592} C_VEL
LIN {X 0,Y 465.247,Z 581.691,A -85,B 0,C 180,E1 -15484.317,E2 -15484.317} C_VEL
LIN {X 0,Y 465.907,Z 578.029,A -85,B 0,C 180,E1 -15486.041,E2 -15486.041} C_VEL
LIN {X 0,Y 466.645,Z 573.765,A -85,B 0,C 180,E1 -15487.476,E2 -15487.476} C_VEL
LIN {X 0,Y 467.781,Z 567.63,A -85,B 0,C 180,E1 -15489.046,E2 -15489.046} C_VEL
LIN {X 0,Y 468.817,Z 560.255,A -85,B 0,C 180,E1 -15490.546,E2 -15490.546} C_VEL
LIN {X 0,Y 469.915,Z 552.488,A -85,B 0,C 180,E1 -15491.827,E2 -15491.827} C_VEL
LIN {X 0,Y 471.066,Z 543.089,A -85,B 0,C 180,E1 -15493.106,E2 -15493.106} C_VEL
LIN {X 0,Y 472.213,Z 532.661,A -85,B 0,C 180,E1 -15494.276,E2 -15494.276} C_VEL
LIN {X 0,Y 473.446,Z 521.174,A -85,B 0,C 180,E1 -15495.334,E2 -15495.334} C_VEL
LIN {X 0,Y 474.636,Z 508.487,A -85,B 0,C 180,E1 -15496.283,E2 -15496.283} C_VEL
LIN {X 0,Y 475.542,Z 494.215,A -85,B 0,C 180,E1 -15497.133,E2 -15497.133} C_VEL
LIN {X 0,Y 476.201,Z 480.339,A -85,B 0,C 180,E1 -15497.771,E2 -15497.771} C_VEL
LIN {X 0,Y 476.633,Z 465.882,A -85,B 0,C 180,E1 -15498.252,E2 -15498.252} C_VEL
LIN {X 0,Y 478.747,Z 412.507,A -85,B 0,C 180,E1 -15499.469,E2 -15499.469} C_VEL
LIN {X 0,Y 480.866,Z 370.711,A -85,B 0,C 180,E1 -15500.44,E2 -15500.44} C_VEL
LIN {X 0,Y 474.525,Z 357.886,A -85,B 0,C 180,E1 -15501.367,E2 -15501.367} C_VEL
LIN {X 0,Y 468.562,Z 347.551,A -85,B 0,C 180,E1 -15502.263,E2 -15502.263} C_VEL
LIN {X 0,Y 466.675,Z 344.252,A -85,B 0,C 180,E1 -15502.564,E2 -15502.564} C_VEL
LIN {X 0,Y 465.07,Z 341.72,A -85,B 0,C 180,E1 -15502.814,E2 -15502.814} C_VEL
LIN {X 0,Y 464.688,Z 340.163,A -85,B 0,C 180,E1 -15502.914,E2 -15502.914} C_VEL
LIN {X 0,Y 464.668,Z 340.165,A -85,B 0,C 180,E1 -15505.922,E2 -15505.922} C_VEL
LIN {X 0,Y 464.674,Z 340.16,A -85,B 0,C 180,E1 -15509.039,E2 -15509.039} C_VEL
LIN {X 0,Y 464.652,Z 340.162,A -85,B 0,C 180,E1 -15512.415,E2 -15512.415} C_VEL
LIN {X 0,Y 464.645,Z 340.159,A -85,B 0,C 180,E1 -15515.507,E2 -15515.507} C_VEL
LIN {X 0,Y 464.615,Z 340.16,A -85,B 0,C 180,E1 -15518.377,E2 -15518.377} C_VEL
LIN {X 0,Y 464.627,Z 340.162,A -85,B 0,C 180,E1 -15521.553,E2 -15521.553} C_VEL
LIN {X 0,Y 464.669,Z 340.159,A -85,B 0,C 180,E1 -15524.888,E2 -15524.888} C_VEL
LIN {X 0,Y 464.632,Z 340.163,A -85,B 0,C 180,E1 -15527.62,E2 -15527.62} C_VEL
LIN {X 0,Y 464.599,Z 340.174,A -85,B 0,C 180,E1 -15530.713,E2 -15530.713} C_VEL
LIN {X 0,Y 464.564,Z 340.175,A -85,B 0,C 180,E1 -15533.983,E2 -15533.983} C_VEL
LIN {X 0,Y 464.623,Z 340.253,A -85,B 0,C 180,E1 -15537.193,E2 -15537.193} C_VEL
LIN {X 0,Y 468.583,Z 356.222,A -85,B 0,C 180,E1 -15539.829,E2 -15539.829} C_VEL
LIN {X 0,Y 471.311,Z 369.013,A -85,B 0,C 180,E1 -15541.845,E2 -15541.845} C_VEL
LIN {X 0,Y 471.367,Z 372.377,A -85,B 0,C 180,E1 -15542.33,E2 -15542.33} C_VEL
LIN {X 0,Y 469.231,Z 396.044,A -85,B 0,C 180,E1 -15545.585,E2 -15545.585} C_VEL
LIN {X 0,Y 468.554,Z 404.474,A -85,B 0,C 180,E1 -15546.735,E2 -15546.735} C_VEL
LIN {X 0,Y 472.4,Z 428.96,A -85,B 0,C 180,E1 -15547.784,E2 -15547.784} C_VEL
LIN {X 0,Y 474.525,Z 445.801,A -85,B 0,C 180,E1 -15548.425,E2 -15548.425} C_VEL
LIN {X 0,Y 476.415,Z 473.278,A -85,B 0,C 180,E1 -15549.313,E2 -15549.313} C_VEL
LIN {X 0,Y 473.203,Z 546.714,A -85,B 0,C 180,E1 -15550.939,E2 -15550.939} C_VEL
LIN {X 0,Y 472.808,Z 563.547,A -85,B 0,C 180,E1 -15551.259,E2 -15551.259} C_VEL
LIN {X 0,Y 471.946,Z 577.093,A -85,B 0,C 180,E1 -15551.672,E2 -15551.672} C_VEL
LIN {X 0,Y 470.755,Z 591.103,A -85,B 0,C 180,E1 -15552.274,E2 -15552.274} C_VEL
LIN {X 0,Y 469.582,Z 603.511,A -85,B 0,C 180,E1 -15552.978,E2 -15552.978} C_VEL
LIN {X 0,Y 468.377,Z 615.416,A -85,B 0,C 180,E1 -15553.827,E2 -15553.827} C_VEL
LIN {X 0,Y 467.016,Z 627.518,A -85,B 0,C 180,E1 -15554.894,E2 -15554.894} C_VEL
LIN {X 0,Y 465.775,Z 638.474,A -85,B 0,C 180,E1 -15556.077,E2 -15556.077} C_VEL
LIN {X 0,Y 464.91,Z 648.197,A -85,B 0,C 180,E1 -15557.326,E2 -15557.326} C_VEL
LIN {X 0,Y 464.332,Z 659.306,A -85,B 0,C 180,E1 -15558.47,E2 -15558.47} C_VEL
LIN {X 0,Y 463.819,Z 669.713,A -85,B 0,C 180,E1 -15559.779,E2 -15559.779} C_VEL
LIN {X 0,Y 463.394,Z 678.313,A -85,B 0,C 180,E1 -15561.087,E2 -15561.087} C_VEL
LIN {X 0,Y 463.087,Z 686.498,A -85,B 0,C 180,E1 -15562.613,E2 -15562.613} C_VEL
LIN {X 0,Y 462.931,Z 692.17,A -85,B 0,C 180,E1 -15563.92,E2 -15563.92} C_VEL
LIN {X 0,Y 462.845,Z 696.769,A -85,B 0,C 180,E1 -15565.225,E2 -15565.225} C_VEL
LIN {X 0,Y 462.751,Z 700.378,A -85,B 0,C 180,E1 -15566.529,E2 -15566.529} C_VEL
LIN {X 0,Y 462.77,Z 702.261,A -85,B 0,C 180,E1 -15567.397,E2 -15567.397} C_VEL
LIN {X 0,Y 462.755,Z 704.837,A -85,B 0,C 180,E1 -15569.133,E2 -15569.133} C_VEL
LIN {X 0,Y 462.739,Z 705.927,A -85,B 0,C 180,E1 -15570.867,E2 -15570.867} C_VEL
LIN {X 0,Y 462.77,Z 705.545,A -85,B 0,C 180,E1 -15572.602,E2 -15572.602} C_VEL
LIN {X 0,Y 462.87,Z 703.703,A -85,B 0,C 180,E1 -15574.339,E2 -15574.339} C_VEL
LIN {X 0,Y 463.164,Z 700.361,A -85,B 0,C 180,E1 -15576.077,E2 -15576.077} C_VEL
LIN {X 0,Y 463.565,Z 695.401,A -85,B 0,C 180,E1 -15577.816,E2 -15577.816} C_VEL
LIN {X 0,Y 464.095,Z 690.593,A -85,B 0,C 180,E1 -15579.118,E2 -15579.118} C_VEL
LIN {X 0,Y 464.955,Z 683.565,A -85,B 0,C 180,E1 -15580.634,E2 -15580.634} C_VEL
LIN {X 0,Y 465.906,Z 674.887,A -85,B 0,C 180,E1 -15582.15,E2 -15582.15} C_VEL
LIN {X 0,Y 466.994,Z 665.82,A -85,B 0,C 180,E1 -15583.443,E2 -15583.443} C_VEL
LIN {X 0,Y 468.35,Z 654.903,A -85,B 0,C 180,E1 -15584.729,E2 -15584.729} C_VEL
LIN {X 0,Y 469.515,Z 643.95,A -85,B 0,C 180,E1 -15585.799,E2 -15585.799} C_VEL
LIN {X 0,Y 470.843,Z 631.984,A -85,B 0,C 180,E1 -15586.752,E2 -15586.752} C_VEL
LIN {X 0,Y 472.075,Z 618.99,A -85,B 0,C 180,E1 -15587.597,E2 -15587.597} C_VEL
LIN {X 0,Y 473.284,Z 604.745,A -85,B 0,C 180,E1 -15588.322,E2 -15588.322} C_VEL
LIN {X 0,Y 474.309,Z 591.252,A -85,B 0,C 180,E1 -15588.835,E2 -15588.835} C_VEL
LIN {X 0,Y 475.193,Z 575.816,A -85,B 0,C 180,E1 -15589.246,E2 -15589.246} C_VEL
LIN {X 0,Y 479.366,Z 490.052,A -85,B 0,C 180,E1 -15591.229,E2 -15591.229} C_VEL
LIN {X 0,Y 480.12,Z 473.481,A -85,B 0,C 180,E1 -15591.638,E2 -15591.638} C_VEL
LIN {X 0,Y 479.273,Z 456.757,A -85,B 0,C 180,E1 -15592.197,E2 -15592.197} C_VEL
LIN {X 0,Y 477.064,Z 436.38,A -85,B 0,C 180,E1 -15593.011,E2 -15593.011} C_VEL
LIN {X 0,Y 476.263,Z 419.523,A -85,B 0,C 180,E1 -15594.088,E2 -15594.088} C_VEL
LIN {X 0,Y 475.266,Z 399.965,A -85,B 0,C 180,E1 -15595.514,E2 -15595.514} C_VEL
LIN {X 0,Y 474.556,Z 387.163,A -85,B 0,C 180,E1 -15596.572,E2 -15596.572} C_VEL
LIN {X 0,Y 474.22,Z 377.651,A -85,B 0,C 180,E1 -15597.414,E2 -15597.414} C_VEL
LIN {X 0,Y 473.872,Z 369.451,A -85,B 0,C 180,E1 -15598.229,E2 -15598.229} C_VEL
LIN {X 0,Y 472.009,Z 359.554,A -85,B 0,C 180,E1 -15599.566,E2 -15599.566} C_VEL
LIN {X 0,Y 470.167,Z 349.833,A -85,B 0,C 180,E1 -15601.117,E2 -15601.117} C_VEL
LIN {X 0,Y 468.19,Z 346.954,A -85,B 0,C 180,E1 -15602.002,E2 -15602.002} C_VEL
LIN {X 0,Y 467.651,Z 345.5,A -85,B 0,C 180,E1 -15602.356,E2 -15602.356} C_VEL
LIN {X 0,Y 465.551,Z 342.966,A -85,B 0,C 180,E1 -15603.383,E2 -15603.383} C_VEL
LIN {X 0,Y 464.581,Z 340.169,A -85,B 0,C 180,E1 -15604.298,E2 -15604.298} C_VEL
LIN {X 0,Y 464.578,Z 340.17,A -85,B 0,C 180,E1 -15607.091,E2 -15607.091} C_VEL
LIN {X 0,Y 464.598,Z 340.171,A -85,B 0,C 180,E1 -15610.412,E2 -15610.412} C_VEL
LIN {X 0,Y 464.632,Z 340.168,A -85,B 0,C 180,E1 -15613.905,E2 -15613.905} C_VEL
LIN {X 0,Y 464.631,Z 340.167,A -85,B 0,C 180,E1 -15616.354,E2 -15616.354} C_VEL
LIN {X 0,Y 464.617,Z 340.329,A -85,B 0,C 180,E1 -15618.651,E2 -15618.651} C_VEL
LIN {X 0,Y 465.659,Z 343.124,A -85,B 0,C 180,E1 -15619.699,E2 -15619.699} C_VEL
LIN {X 0,Y 466.873,Z 344.744,A -85,B 0,C 180,E1 -15620.433,E2 -15620.433} C_VEL
LIN {X 0,Y 467.7,Z 347.063,A -85,B 0,C 180,E1 -15621.148,E2 -15621.148} C_VEL
LIN {X 0,Y 469.458,Z 350.503,A -85,B 0,C 180,E1 -15622.285,E2 -15622.285} C_VEL
LIN {X 0,Y 472.477,Z 357.321,A -85,B 0,C 180,E1 -15624.179,E2 -15624.179} C_VEL
LIN {X 0,Y 475.692,Z 366.052,A -85,B 0,C 180,E1 -15626.225,E2 -15626.225} C_VEL
LIN {X 0,Y 478.579,Z 375.85,A -85,B 0,C 180,E1 -15628.204,E2 -15628.204} C_VEL
LIN {X 0,Y 480.309,Z 383.267,A -85,B 0,C 180,E1 -15629.555,E2 -15629.555} C_VEL
LIN {X 0,Y 481.038,Z 388,A -85,B 0,C 180,E1 -15630.325,E2 -15630.325} C_VEL
LIN {X 0,Y 478.617,Z 409.064,A -85,B 0,C 180,E1 -15633.02,E2 -15633.02} C_VEL
LIN {X 0,Y 475.609,Z 437.377,A -85,B 0,C 180,E1 -15636.57,E2 -15636.57} C_VEL
LIN {X 0,Y 475.479,Z 440.131,A -85,B 0,C 180,E1 -15636.879,E2 -15636.879} C_VEL
LIN {X 0,Y 478.894,Z 458.112,A -85,B 0,C 180,E1 -15637.72,E2 -15637.72} C_VEL
LIN {X 0,Y 480.701,Z 472.155,A -85,B 0,C 180,E1 -15638.278,E2 -15638.278} C_VEL
LIN {X 0,Y 476.658,Z 553.942,A -85,B 0,C 180,E1 -15640.171,E2 -15640.171} C_VEL
LIN {X 0,Y 475.215,Z 583.162,A -85,B 0,C 180,E1 -15640.851,E2 -15640.851} C_VEL
LIN {X 0,Y 474.197,Z 596.839,A -85,B 0,C 180,E1 -15641.316,E2 -15641.316} C_VEL
LIN {X 0,Y 472.965,Z 611.393,A -85,B 0,C 180,E1 -15641.992,E2 -15641.992} C_VEL
LIN {X 0,Y 471.724,Z 625.316,A -85,B 0,C 180,E1 -15642.836,E2 -15642.836} C_VEL
LIN {X 0,Y 470.329,Z 637.94,A -85,B 0,C 180,E1 -15643.786,E2 -15643.786} C_VEL
LIN {X 0,Y 469,Z 649.471,A -85,B 0,C 180,E1 -15644.849,E2 -15644.849} C_VEL
LIN {X 0,Y 467.881,Z 659.148,A -85,B 0,C 180,E1 -15645.92,E2 -15645.92} C_VEL
LIN {X 0,Y 466.559,Z 669.14,A -85,B 0,C 180,E1 -15647.237,E2 -15647.237} C_VEL
LIN {X 0,Y 465.606,Z 678.304,A -85,B 0,C 180,E1 -15648.722,E2 -15648.722} C_VEL
LIN {X 0,Y 464.695,Z 684.91,A -85,B 0,C 180,E1 -15650.018,E2 -15650.018} C_VEL
LIN {X 0,Y 464.055,Z 690.379,A -85,B 0,C 180,E1 -15651.319,E2 -15651.319} C_VEL
LIN {X 0,Y 463.496,Z 694.851,A -85,B 0,C 180,E1 -15652.62,E2 -15652.62} C_VEL
LIN {X 0,Y 463.126,Z 698.38,A -85,B 0,C 180,E1 -15653.923,E2 -15653.923} C_VEL
LIN {X 0,Y 462.87,Z 701.707,A -85,B 0,C 180,E1 -15655.661,E2 -15655.661} C_VEL
LIN {X 0,Y 462.695,Z 703.54,A -85,B 0,C 180,E1 -15657.397,E2 -15657.397} C_VEL
LIN {X 0,Y 462.658,Z 703.932,A -85,B 0,C 180,E1 -15659.133,E2 -15659.133} C_VEL
LIN {X 0,Y 462.657,Z 702.871,A -85,B 0,C 180,E1 -15660.868,E2 -15660.868} C_VEL
LIN {X 0,Y 462.689,Z 700.344,A -85,B 0,C 180,E1 -15662.603,E2 -15662.603} C_VEL
LIN {X 0,Y 462.734,Z 697.407,A -85,B 0,C 180,E1 -15663.906,E2 -15663.906} C_VEL
LIN {X 0,Y 462.825,Z 693.573,A -85,B 0,C 180,E1 -15665.21,E2 -15665.21} C_VEL
LIN {X 0,Y 462.947,Z 688.755,A -85,B 0,C 180,E1 -15666.516,E2 -15666.516} C_VEL
LIN {X 0,Y 463.233,Z 681.7,A -85,B 0,C 180,E1 -15668.04,E2 -15668.04} C_VEL
LIN {X 0,Y 463.693,Z 672.915,A -85,B 0,C 180,E1 -15669.565,E2 -15669.565} C_VEL
LIN {X 0,Y 464.185,Z 663.945,A -85,B 0,C 180,E1 -15670.843,E2 -15670.843} C_VEL
LIN {X 0,Y 464.679,Z 654.566,A -85,B 0,C 180,E1 -15671.962,E2 -15671.962} C_VEL
LIN {X 0,Y 465.349,Z 642.516,A -85,B 0,C 180,E1 -15673.16,E2 -15673.16} C_VEL
LIN {X 0,Y 466.023,Z 630.42,A -85,B 0,C 180,E1 -15674.137,E2 -15674.137} C_VEL
LIN {X 0,Y 466.795,Z 617.197,A -85,B 0,C 180,E1 -15675.002,E2 -15675.002} C_VEL
LIN {X 0,Y 467.306,Z 603.538,A -85,B 0,C 180,E1 -15675.709,E2 -15675.709} C_VEL
LIN {X 0,Y 467.836,Z 588.95,A -85,B 0,C 180,E1 -15676.276,E2 -15676.276} C_VEL
LIN {X 0,Y 468.309,Z 573.944,A -85,B 0,C 180,E1 -15676.669,E2 -15676.669} C_VEL
LIN {X 0,Y 470.616,Z 468.515,A -85,B 0,C 180,E1 -15678.776,E2 -15678.776} C_VEL
LIN {X 0,Y 467.742,Z 439.432,A -85,B 0,C 180,E1 -15679.481,E2 -15679.481} C_VEL
LIN {X 0,Y 469.272,Z 409.247,A -85,B 0,C 180,E1 -15683.068,E2 -15683.068} C_VEL
LIN {X 0,Y 470.674,Z 384.303,A -85,B 0,C 180,E1 -15686.041,E2 -15686.041} C_VEL
LIN {X 0,Y 471.35,Z 370.682,A -85,B 0,C 180,E1 -15687.671,E2 -15687.671} C_VEL
LIN {X 0,Y 468.333,Z 356.169,A -85,B 0,C 180,E1 -15689.575,E2 -15689.575} C_VEL
LIN {X 0,Y 464.685,Z 340.16,A -85,B 0,C 180,E1 -15691.728,E2 -15691.728} C_VEL
LIN {X 0,Y 464.652,Z 340.163,A -85,B 0,C 180,E1 -15694.949,E2 -15694.949} C_VEL
LIN {X 0,Y 464.615,Z 340.164,A -85,B 0,C 180,E1 -15698.179,E2 -15698.179} C_VEL
LIN {X 0,Y 464.663,Z 340.158,A -85,B 0,C 180,E1 -15700.406,E2 -15700.406} C_VEL
LIN {X 0,Y 464.651,Z 340.159,A -85,B 0,C 180,E1 -15703.903,E2 -15703.903} C_VEL
LIN {X 0,Y 464.649,Z 340.161,A -85,B 0,C 180,E1 -15706.352,E2 -15706.352} C_VEL
LIN {X 0,Y 464.666,Z 340.158,A -85,B 0,C 180,E1 -15709.595,E2 -15709.595} C_VEL
LIN {X 0,Y 464.636,Z 340.165,A -85,B 0,C 180,E1 -15713.034,E2 -15713.034} C_VEL
LIN {X 0,Y 464.673,Z 340.158,A -85,B 0,C 180,E1 -15716.101,E2 -15716.101} C_VEL
LIN {X 0,Y 464.658,Z 340.159,A -85,B 0,C 180,E1 -15719.232,E2 -15719.232} C_VEL
LIN {X 0,Y 464.682,Z 340.16,A -85,B 0,C 180,E1 -15722.142,E2 -15722.142} C_VEL
LIN {X 0,Y 464.656,Z 340.159,A -85,B 0,C 180,E1 -15725.034,E2 -15725.034} C_VEL
LIN {X 0,Y 464.68,Z 340.159,A -85,B 0,C 180,E1 -15727.862,E2 -15727.862} C_VEL
LIN {X 0,Y 464.684,Z 340.158,A -85,B 0,C 180,E1 -15730.633,E2 -15730.633} C_VEL
LIN {X 0,Y 464.673,Z 340.157,A -85,B 0,C 180,E1 -15733.357,E2 -15733.357} C_VEL
LIN {X 0,Y 464.739,Z 340.158,A -85,B 0,C 180,E1 -15735.175,E2 -15735.175} C_VEL
LIN {X 0,Y 470.019,Z 354.513,A -85,B 0,C 180,E1 -15735.62,E2 -15735.62} C_VEL
LIN {X 0,Y 472.655,Z 362.246,A -85,B 0,C 180,E1 -15735.846,E2 -15735.846} C_VEL
LIN {X 0,Y 471.544,Z 455.277,A -85,B 0,C 180,E1 -15737.262,E2 -15737.262} C_VEL
LIN {X 0,Y 471.425,Z 469.334,A -85,B 0,C 180,E1 -15737.586,E2 -15737.586} C_VEL
LIN {X 0,Y 471.121,Z 483.638,A -85,B 0,C 180,E1 -15738.095,E2 -15738.095} C_VEL
LIN {X 0,Y 470.567,Z 496.79,A -85,B 0,C 180,E1 -15738.734,E2 -15738.734} C_VEL
LIN {X 0,Y 469.885,Z 510.288,A -85,B 0,C 180,E1 -15739.587,E2 -15739.587} C_VEL
LIN {X 0,Y 469.195,Z 522.331,A -85,B 0,C 180,E1 -15740.548,E2 -15740.548} C_VEL
LIN {X 0,Y 468.344,Z 533.273,A -85,B 0,C 180,E1 -15741.615,E2 -15741.615} C_VEL
LIN {X 0,Y 467.378,Z 544.037,A -85,B 0,C 180,E1 -15742.898,E2 -15742.898} C_VEL
LIN {X 0,Y 466.515,Z 552.937,A -85,B 0,C 180,E1 -15744.183,E2 -15744.183} C_VEL
LIN {X 0,Y 465.795,Z 561.432,A -85,B 0,C 180,E1 -15745.688,E2 -15745.688} C_VEL
LIN {X 0,Y 465.195,Z 567.427,A -85,B 0,C 180,E1 -15746.979,E2 -15746.979} C_VEL
LIN {X 0,Y 464.612,Z 573.798,A -85,B 0,C 180,E1 -15748.704,E2 -15748.704} C_VEL
LIN {X 0,Y 464.271,Z 578.565,A -85,B 0,C 180,E1 -15750.432,E2 -15750.432} C_VEL
LIN {X 0,Y 464.148,Z 581.826,A -85,B 0,C 180,E1 -15752.166,E2 -15752.166} C_VEL
LIN {X 0,Y 463.476,Z 582.922,A -85,B 0,C 180,E1 -15752.879,E2 -15752.879} C_VEL
LIN {X 0,Y 460.559,Z 584.339,A -85,B 0,C 180,E1 -15754.041,E2 -15754.041} C_VEL
LIN {X 0,Y 458.125,Z 585.059,A -85,B 0,C 180,E1 -15754.984,E2 -15754.984} C_VEL
LIN {X 0,Y 457.126,Z 585.296,A -85,B 0,C 180,E1 -15755.715,E2 -15755.715} C_VEL
LIN {X 0,Y 457.071,Z 585.234,A -85,B 0,C 180,E1 -15755.962,E2 -15755.962} C_VEL
LIN {X 0,Y 457.176,Z 584.91,A -85,B 0,C 180,E1 -15757.041,E2 -15757.041} C_VEL
LIN {X 0,Y 457.439,Z 583.287,A -85,B 0,C 180,E1 -15758.808,E2 -15758.808} C_VEL
LIN {X 0,Y 457.919,Z 580.313,A -85,B 0,C 180,E1 -15760.577,E2 -15760.577} C_VEL
LIN {X 0,Y 458.641,Z 575.884,A -85,B 0,C 180,E1 -15762.346,E2 -15762.346} C_VEL
LIN {X 0,Y 459.492,Z 569.811,A -85,B 0,C 180,E1 -15764.117,E2 -15764.117} C_VEL
LIN {X 0,Y 460.439,Z 563.005,A -85,B 0,C 180,E1 -15765.666,E2 -15765.666} C_VEL
LIN {X 0,Y 461.57,Z 554.794,A -85,B 0,C 180,E1 -15767.167,E2 -15767.167} C_VEL
LIN {X 0,Y 462.72,Z 545.632,A -85,B 0,C 180,E1 -15768.536,E2 -15768.536} C_VEL
LIN {X 0,Y 463.88,Z 534.822,A -85,B 0,C 180,E1 -15769.861,E2 -15769.861} C_VEL
LIN {X 0,Y 464.921,Z 524.281,A -85,B 0,C 180,E1 -15770.918,E2 -15770.918} C_VEL
LIN {X 0,Y 466.1,Z 511.553,A -85,B 0,C 180,E1 -15771.951,E2 -15771.951} C_VEL
LIN {X 0,Y 466.96,Z 499.731,A -85,B 0,C 180,E1 -15772.722,E2 -15772.722} C_VEL
LIN {X 0,Y 467.431,Z 488.029,A -85,B 0,C 180,E1 -15773.339,E2 -15773.339} C_VEL
LIN {X 0,Y 467.901,Z 474.173,A -85,B 0,C 180,E1 -15773.883,E2 -15773.883} C_VEL
LIN {X 0,Y 468.19,Z 460.956,A -85,B 0,C 180,E1 -15774.236,E2 -15774.236} C_VEL
LIN {X 0,Y 469.104,Z 402.12,A -85,B 0,C 180,E1 -15775.163,E2 -15775.163} C_VEL
LIN {X 0,Y 469.573,Z 368.642,A -85,B 0,C 180,E1 -15775.685,E2 -15775.685} C_VEL
LIN {X 0,Y 460.072,Z 346.933,A -85,B 0,C 180,E1 -15776.562,E2 -15776.562} C_VEL
LIN {X 0,Y 457.749,Z 341.819,A -85,B 0,C 180,E1 -15776.78,E2 -15776.78} C_VEL
LIN {X 0,Y 457.605,Z 341.048,A -85,B 0,C 180,E1 -15776.828,E2 -15776.828} C_VEL
LIN {X 0,Y 457.627,Z 341.04,A -85,B 0,C 180,E1 -15779.327,E2 -15779.327} C_VEL
LIN {X 0,Y 457.526,Z 341.051,A -85,B 0,C 180,E1 -15782.646,E2 -15782.646} C_VEL
LIN {X 0,Y 457.543,Z 341.05,A -85,B 0,C 180,E1 -15785.77,E2 -15785.77} C_VEL
LIN {X 0,Y 457.557,Z 341.047,A -85,B 0,C 180,E1 -15788.877,E2 -15788.877} C_VEL
LIN {X 0,Y 457.575,Z 341.047,A -85,B 0,C 180,E1 -15792.341,E2 -15792.341} C_VEL
LIN {X 0,Y 457.613,Z 341.036,A -85,B 0,C 180,E1 -15795.243,E2 -15795.243} C_VEL
LIN {X 0,Y 457.59,Z 341.041,A -85,B 0,C 180,E1 -15798.596,E2 -15798.596} C_VEL
LIN {X 0,Y 457.554,Z 341.04,A -85,B 0,C 180,E1 -15801.328,E2 -15801.328} C_VEL
LIN {X 0,Y 457.563,Z 341.023,A -85,B 0,C 180,E1 -15804.429,E2 -15804.429} C_VEL
LIN {X 0,Y 457.569,Z 341.045,A -85,B 0,C 180,E1 -15807.603,E2 -15807.603} C_VEL
LIN {X 0,Y 457.631,Z 341.032,A -85,B 0,C 180,E1 -15810.743,E2 -15810.743} C_VEL
LIN {X 0,Y 457.612,Z 341.033,A -85,B 0,C 180,E1 -15813.647,E2 -15813.647} C_VEL
LIN {X 0,Y 457.576,Z 341.042,A -85,B 0,C 180,E1 -15816.703,E2 -15816.703} C_VEL
LIN {X 0,Y 457.635,Z 341.043,A -85,B 0,C 180,E1 -15820.058,E2 -15820.058} C_VEL
LIN {X 0,Y 463.32,Z 360.524,A -85,B 0,C 180,E1 -15820.642,E2 -15820.642} C_VEL
LIN {X 0,Y 461.362,Z 459.619,A -85,B 0,C 180,E1 -15822.652,E2 -15822.652} C_VEL
LIN {X 0,Y 461.186,Z 475.505,A -85,B 0,C 180,E1 -15823.171,E2 -15823.171} C_VEL
LIN {X 0,Y 460.758,Z 490.127,A -85,B 0,C 180,E1 -15823.836,E2 -15823.836} C_VEL
LIN {X 0,Y 460.204,Z 504.06,A -85,B 0,C 180,E1 -15824.665,E2 -15824.665} C_VEL
LIN {X 0,Y 459.672,Z 517.428,A -85,B 0,C 180,E1 -15825.663,E2 -15825.663} C_VEL
LIN {X 0,Y 459.023,Z 529.455,A -85,B 0,C 180,E1 -15826.768,E2 -15826.768} C_VEL
LIN {X 0,Y 458.629,Z 540.18,A -85,B 0,C 180,E1 -15827.965,E2 -15827.965} C_VEL
LIN {X 0,Y 458.062,Z 551.007,A -85,B 0,C 180,E1 -15829.426,E2 -15829.426} C_VEL
LIN {X 0,Y 457.575,Z 560.304,A -85,B 0,C 180,E1 -15830.972,E2 -15830.972} C_VEL
LIN {X 0,Y 457.215,Z 567.79,A -85,B 0,C 180,E1 -15832.518,E2 -15832.518} C_VEL
LIN {X 0,Y 457.033,Z 573.01,A -85,B 0,C 180,E1 -15833.841,E2 -15833.841} C_VEL
LIN {X 0,Y 456.929,Z 578.418,A -85,B 0,C 180,E1 -15835.604,E2 -15835.604} C_VEL
LIN {X 0,Y 456.958,Z 582.242,A -85,B 0,C 180,E1 -15837.364,E2 -15837.364} C_VEL
LIN {X 0,Y 456.978,Z 584.54,A -85,B 0,C 180,E1 -15839.122,E2 -15839.122} C_VEL
LIN {X 0,Y 457.188,Z 585.404,A -85,B 0,C 180,E1 -15840.878,E2 -15840.878} C_VEL
LIN {X 0,Y 457.559,Z 584.844,A -85,B 0,C 180,E1 -15842.632,E2 -15842.632} C_VEL
LIN {X 0,Y 458.26,Z 582.833,A -85,B 0,C 180,E1 -15844.383,E2 -15844.383} C_VEL
LIN {X 0,Y 458.965,Z 579.32,A -85,B 0,C 180,E1 -15846.132,E2 -15846.132} C_VEL
LIN {X 0,Y 459.645,Z 575.664,A -85,B 0,C 180,E1 -15847.442,E2 -15847.442} C_VEL
LIN {X 0,Y 460.618,Z 570.968,A -85,B 0,C 180,E1 -15848.746,E2 -15848.746} C_VEL
LIN {X 0,Y 461.737,Z 564.209,A -85,B 0,C 180,E1 -15850.267,E2 -15850.267} C_VEL
LIN {X 0,Y 462.787,Z 557.061,A -85,B 0,C 180,E1 -15851.569,E2 -15851.569} C_VEL
LIN {X 0,Y 464.001,Z 548.429,A -85,B 0,C 180,E1 -15852.865,E2 -15852.865} C_VEL
LIN {X 0,Y 465.202,Z 538,A -85,B 0,C 180,E1 -15854.162,E2 -15854.162} C_VEL
LIN {X 0,Y 466.596,Z 526.287,A -85,B 0,C 180,E1 -15855.342,E2 -15855.342} C_VEL
LIN {X 0,Y 467.916,Z 514.087,A -85,B 0,C 180,E1 -15856.336,E2 -15856.336} C_VEL
LIN {X 0,Y 469.036,Z 500.104,A -85,B 0,C 180,E1 -15857.251,E2 -15857.251} C_VEL
LIN {X 0,Y 469.799,Z 486.291,A -85,B 0,C 180,E1 -15857.965,E2 -15857.965} C_VEL
LIN {X 0,Y 470.41,Z 472.156,A -85,B 0,C 180,E1 -15858.502,E2 -15858.502} C_VEL
LIN {X 0,Y 470.821,Z 454.889,A -85,B 0,C 180,E1 -15858.964,E2 -15858.964} C_VEL
LIN {X 0,Y 475.012,Z 373.196,A -85,B 0,C 180,E1 -15860.873,E2 -15860.873} C_VEL
LIN {X 0,Y 468.953,Z 361.075,A -85,B 0,C 180,E1 -15861.796,E2 -15861.796} C_VEL
LIN {X 0,Y 463.69,Z 351.82,A -85,B 0,C 180,E1 -15862.629,E2 -15862.629} C_VEL
LIN {X 0,Y 460.213,Z 345.9,A -85,B 0,C 180,E1 -15863.197,E2 -15863.197} C_VEL
LIN {X 0,Y 458.178,Z 343.119,A -85,B 0,C 180,E1 -15863.532,E2 -15863.532} C_VEL
LIN {X 0,Y 457.61,Z 341.045,A -85,B 0,C 180,E1 -15863.69,E2 -15863.69} C_VEL
LIN {X 0,Y 457.645,Z 341.039,A -85,B 0,C 180,E1 -15866.35,E2 -15866.35} C_VEL
LIN {X 0,Y 457.629,Z 341.039,A -85,B 0,C 180,E1 -15869.327,E2 -15869.327} C_VEL
LIN {X 0,Y 457.63,Z 341.037,A -85,B 0,C 180,E1 -15872.666,E2 -15872.666} C_VEL
LIN {X 0,Y 457.613,Z 341.035,A -85,B 0,C 180,E1 -15875.782,E2 -15875.782} C_VEL
LIN {X 0,Y 457.581,Z 341.035,A -85,B 0,C 180,E1 -15878.874,E2 -15878.874} C_VEL
LIN {X 0,Y 457.584,Z 341.035,A -85,B 0,C 180,E1 -15882.34,E2 -15882.34} C_VEL
LIN {X 0,Y 457.612,Z 341.041,A -85,B 0,C 180,E1 -15885.243,E2 -15885.243} C_VEL
LIN {X 0,Y 457.588,Z 341.043,A -85,B 0,C 180,E1 -15888.595,E2 -15888.595} C_VEL
LIN {X 0,Y 457.552,Z 341.046,A -85,B 0,C 180,E1 -15891.328,E2 -15891.328} C_VEL
LIN {X 0,Y 457.538,Z 341.05,A -85,B 0,C 180,E1 -15894.427,E2 -15894.427} C_VEL
LIN {X 0,Y 457.563,Z 341.095,A -85,B 0,C 180,E1 -15896.843,E2 -15896.843} C_VEL
LIN {X 0,Y 461.404,Z 356.44,A -85,B 0,C 180,E1 -15899.433,E2 -15899.433} C_VEL
LIN {X 0,Y 464.361,Z 370.128,A -85,B 0,C 180,E1 -15901.631,E2 -15901.631} C_VEL
LIN {X 0,Y 464.56,Z 373.498,A -85,B 0,C 180,E1 -15902.134,E2 -15902.134} C_VEL
LIN {X 0,Y 462.197,Z 398.819,A -85,B 0,C 180,E1 -15905.668,E2 -15905.668} C_VEL
LIN {X 0,Y 462.029,Z 401.711,A -85,B 0,C 180,E1 -15906.031,E2 -15906.031} C_VEL
LIN {X 0,Y 466.105,Z 427.164,A -85,B 0,C 180,E1 -15907.193,E2 -15907.193} C_VEL
LIN {X 0,Y 468.556,Z 447.059,A -85,B 0,C 180,E1 -15907.986,E2 -15907.986} C_VEL
LIN {X 0,Y 470.313,Z 473.938,A -85,B 0,C 180,E1 -15908.88,E2 -15908.88} C_VEL
LIN {X 0,Y 466.392,Z 556.524,A -85,B 0,C 180,E1 -15910.792,E2 -15910.792} C_VEL
LIN {X 0,Y 465.524,Z 572.615,A -85,B 0,C 180,E1 -15911.239,E2 -15911.239} C_VEL
LIN {X 0,Y 464.361,Z 586.927,A -85,B 0,C 180,E1 -15911.815,E2 -15911.815} C_VEL
LIN {X 0,Y 463.131,Z 599.754,A -85,B 0,C 180,E1 -15912.507,E2 -15912.507} C_VEL
LIN {X 0,Y 461.788,Z 612.232,A -85,B 0,C 180,E1 -15913.363,E2 -15913.363} C_VEL
LIN {X 0,Y 460.404,Z 624.848,A -85,B 0,C 180,E1 -15914.446,E2 -15914.446} C_VEL
LIN {X 0,Y 459.056,Z 636.148,A -85,B 0,C 180,E1 -15915.644,E2 -15915.644} C_VEL
LIN {X 0,Y 458.049,Z 646.317,A -85,B 0,C 180,E1 -15916.964,E2 -15916.964} C_VEL
LIN {X 0,Y 457.766,Z 649.649,A -85,B 0,C 180,E1 -15917.406,E2 -15917.406} C_VEL
LIN {X 0,Y 457.206,Z 659.994,A -85,B 0,C 180,E1 -15918.512,E2 -15918.512} C_VEL
LIN {X 0,Y 456.689,Z 670.277,A -85,B 0,C 180,E1 -15919.841,E2 -15919.841} C_VEL
LIN {X 0,Y 456.282,Z 678.781,A -85,B 0,C 180,E1 -15921.169,E2 -15921.169} C_VEL
LIN {X 0,Y 455.983,Z 686.886,A -85,B 0,C 180,E1 -15922.719,E2 -15922.719} C_VEL
LIN {X 0,Y 455.832,Z 693.337,A -85,B 0,C 180,E1 -15924.268,E2 -15924.268} C_VEL
LIN {X 0,Y 455.737,Z 697.671,A -85,B 0,C 180,E1 -15925.592,E2 -15925.592} C_VEL
LIN {X 0,Y 455.69,Z 701.994,A -85,B 0,C 180,E1 -15927.357,E2 -15927.357} C_VEL
LIN {X 0,Y 455.681,Z 703.544,A -85,B 0,C 180,E1 -15928.238,E2 -15928.238} C_VEL
LIN {X 0,Y 455.656,Z 705.475,A -85,B 0,C 180,E1 -15930,E2 -15930} C_VEL
LIN {X 0,Y 455.681,Z 705.927,A -85,B 0,C 180,E1 -15931.762,E2 -15931.762} C_VEL
LIN {X 0,Y 455.738,Z 704.909,A -85,B 0,C 180,E1 -15933.525,E2 -15933.525} C_VEL
LIN {X 0,Y 455.898,Z 702.432,A -85,B 0,C 180,E1 -15935.289,E2 -15935.289} C_VEL
LIN {X 0,Y 456.301,Z 698.435,A -85,B 0,C 180,E1 -15937.054,E2 -15937.054} C_VEL
LIN {X 0,Y 456.888,Z 692.752,A -85,B 0,C 180,E1 -15938.819,E2 -15938.819} C_VEL
LIN {X 0,Y 457.698,Z 686.319,A -85,B 0,C 180,E1 -15940.359,E2 -15940.359} C_VEL
LIN {X 0,Y 458.684,Z 678.652,A -85,B 0,C 180,E1 -15941.832,E2 -15941.832} C_VEL
LIN {X 0,Y 459.737,Z 669.946,A -85,B 0,C 180,E1 -15943.211,E2 -15943.211} C_VEL
LIN {X 0,Y 461.13,Z 659.895,A -85,B 0,C 180,E1 -15944.515,E2 -15944.515} C_VEL
LIN {X 0,Y 462.372,Z 648.833,A -85,B 0,C 180,E1 -15945.711,E2 -15945.711} C_VEL
LIN {X 0,Y 463.872,Z 636.564,A -85,B 0,C 180,E1 -15946.785,E2 -15946.785} C_VEL
LIN {X 0,Y 465.321,Z 622.985,A -85,B 0,C 180,E1 -15947.747,E2 -15947.747} C_VEL
LIN {X 0,Y 466.557,Z 609.842,A -85,B 0,C 180,E1 -15948.491,E2 -15948.491} C_VEL
LIN {X 0,Y 467.794,Z 595.111,A -85,B 0,C 180,E1 -15949.12,E2 -15949.12} C_VEL
LIN {X 0,Y 468.777,Z 580.101,A -85,B 0,C 180,E1 -15949.572,E2 -15949.572} C_VEL
LIN {X 0,Y 473.551,Z 489.349,A -85,B 0,C 180,E1 -15951.727,E2 -15951.727} C_VEL
LIN {X 0,Y 474.263,Z 473.959,A -85,B 0,C 180,E1 -15952.121,E2 -15952.121} C_VEL
LIN {X 0,Y 473.433,Z 457.037,A -85,B 0,C 180,E1 -15952.709,E2 -15952.709} C_VEL
LIN {X 0,Y 471.227,Z 435.888,A -85,B 0,C 180,E1 -15953.604,E2 -15953.604} C_VEL
LIN {X 0,Y 470.442,Z 416.21,A -85,B 0,C 180,E1 -15954.941,E2 -15954.941} C_VEL
LIN {X 0,Y 469.791,Z 399.836,A -85,B 0,C 180,E1 -15956.218,E2 -15956.218} C_VEL
LIN {X 0,Y 469.445,Z 390.161,A -85,B 0,C 180,E1 -15957.046,E2 -15957.046} C_VEL
LIN {X 0,Y 469.261,Z 380.896,A -85,B 0,C 180,E1 -15957.886,E2 -15957.886} C_VEL
LIN {X 0,Y 468.96,Z 372.993,A -85,B 0,C 180,E1 -15958.686,E2 -15958.686} C_VEL
LIN {X 0,Y 467.488,Z 364.295,A -85,B 0,C 180,E1 -15959.896,E2 -15959.896} C_VEL
LIN {X 0,Y 466.214,Z 356.746,A -85,B 0,C 180,E1 -15961.088,E2 -15961.088} C_VEL
LIN {X 0,Y 465.711,Z 354.981,A -85,B 0,C 180,E1 -15961.448,E2 -15961.448} C_VEL
LIN {X 0,Y 463.259,Z 350.744,A -85,B 0,C 180,E1 -15962.704,E2 -15962.704} C_VEL
LIN {X 0,Y 461.141,Z 347.716,A -85,B 0,C 180,E1 -15963.865,E2 -15963.865} C_VEL
LIN {X 0,Y 460.762,Z 346.589,A -85,B 0,C 180,E1 -15964.227,E2 -15964.227} C_VEL
LIN {X 0,Y 458.333,Z 343.533,A -85,B 0,C 180,E1 -15965.907,E2 -15965.907} C_VEL
LIN {X 0,Y 457.549,Z 341.045,A -85,B 0,C 180,E1 -15967.167,E2 -15967.167} C_VEL
LIN {X 0,Y 457.549,Z 341.045,A -85,B 0,C 180,E1 -15970.055,E2 -15970.055} C_VEL
LIN {X 0,Y 457.563,Z 341.048,A -85,B 0,C 180,E1 -15972.711,E2 -15972.711} C_VEL
LIN {X 0,Y 457.615,Z 341.134,A -85,B 0,C 180,E1 -15975.9,E2 -15975.9} C_VEL
LIN {X 0,Y 459.031,Z 344.579,A -85,B 0,C 180,E1 -15977.825,E2 -15977.825} C_VEL
LIN {X 0,Y 460.102,Z 345.94,A -85,B 0,C 180,E1 -15978.623,E2 -15978.623} C_VEL
LIN {X 0,Y 461.278,Z 348.8,A -85,B 0,C 180,E1 -15979.772,E2 -15979.772} C_VEL
LIN {X 0,Y 462.367,Z 350.799,A -85,B 0,C 180,E1 -15980.588,E2 -15980.588} C_VEL
LIN {X 0,Y 464.72,Z 355.95,A -85,B 0,C 180,E1 -15982.307,E2 -15982.307} C_VEL
LIN {X 0,Y 467.63,Z 362.857,A -85,B 0,C 180,E1 -15984.256,E2 -15984.256} C_VEL
LIN {X 0,Y 470.424,Z 370.983,A -85,B 0,C 180,E1 -15986.184,E2 -15986.184} C_VEL
LIN {X 0,Y 472.804,Z 379.517,A -85,B 0,C 180,E1 -15987.955,E2 -15987.955} C_VEL
LIN {X 0,Y 474.618,Z 387.475,A -85,B 0,C 180,E1 -15989.428,E2 -15989.428} C_VEL
LIN {X 0,Y 475.04,Z 390.309,A -85,B 0,C 180,E1 -15989.912,E2 -15989.912} C_VEL
LIN {X 0,Y 474.369,Z 397.16,A -85,B 0,C 180,E1 -15990.839,E2 -15990.839} C_VEL
LIN {X 0,Y 471.105,Z 423.534,A -85,B 0,C 180,E1 -15994.222,E2 -15994.222} C_VEL
LIN {X 0,Y 469.427,Z 439.992,A -85,B 0,C 180,E1 -15996.285,E2 -15996.285} C_VEL
LIN {X 0,Y 472.854,Z 458.025,A -85,B 0,C 180,E1 -15997.178,E2 -15997.178} C_VEL
LIN {X 0,Y 474.86,Z 473.594,A -85,B 0,C 180,E1 -15997.826,E2 -15997.826} C_VEL
LIN {X 0,Y 470.526,Z 554.776,A -85,B 0,C 180,E1 -15999.751,E2 -15999.751} C_VEL
LIN {X 0,Y 468.989,Z 583.662,A -85,B 0,C 180,E1 -16000.444,E2 -16000.444} C_VEL
LIN {X 0,Y 467.876,Z 597.748,A -85,B 0,C 180,E1 -16000.941,E2 -16000.941} C_VEL
LIN {X 0,Y 466.572,Z 612.025,A -85,B 0,C 180,E1 -16001.623,E2 -16001.623} C_VEL
LIN {X 0,Y 465.265,Z 625.781,A -85,B 0,C 180,E1 -16002.477,E2 -16002.477} C_VEL
LIN {X 0,Y 463.785,Z 638.279,A -85,B 0,C 180,E1 -16003.437,E2 -16003.437} C_VEL
LIN {X 0,Y 462.271,Z 650.749,A -85,B 0,C 180,E1 -16004.623,E2 -16004.623} C_VEL
LIN {X 0,Y 461.082,Z 660.237,A -85,B 0,C 180,E1 -16005.708,E2 -16005.708} C_VEL
LIN {X 0,Y 459.698,Z 670.137,A -85,B 0,C 180,E1 -16007.058,E2 -16007.058} C_VEL
LIN {X 0,Y 458.692,Z 679.047,A -85,B 0,C 180,E1 -16008.55,E2 -16008.55} C_VEL
LIN {X 0,Y 457.733,Z 685.533,A -85,B 0,C 180,E1 -16009.865,E2 -16009.865} C_VEL
LIN {X 0,Y 457.063,Z 690.875,A -85,B 0,C 180,E1 -16011.185,E2 -16011.185} C_VEL
LIN {X 0,Y 456.342,Z 696.511,A -85,B 0,C 180,E1 -16012.947,E2 -16012.947} C_VEL
LIN {X 0,Y 455.888,Z 700.482,A -85,B 0,C 180,E1 -16014.711,E2 -16014.711} C_VEL
LIN {X 0,Y 455.663,Z 702.941,A -85,B 0,C 180,E1 -16016.475,E2 -16016.475} C_VEL
LIN {X 0,Y 455.593,Z 703.958,A -85,B 0,C 180,E1 -16018.238,E2 -16018.238} C_VEL
LIN {X 0,Y 455.584,Z 703.526,A -85,B 0,C 180,E1 -16020,E2 -16020} C_VEL
LIN {X 0,Y 455.593,Z 701.637,A -85,B 0,C 180,E1 -16021.762,E2 -16021.762} C_VEL
LIN {X 0,Y 455.633,Z 698.206,A -85,B 0,C 180,E1 -16023.526,E2 -16023.526} C_VEL
LIN {X 0,Y 455.743,Z 693.144,A -85,B 0,C 180,E1 -16025.291,E2 -16025.291} C_VEL
LIN {X 0,Y 455.879,Z 688.199,A -85,B 0,C 180,E1 -16026.617,E2 -16026.617} C_VEL
LIN {X 0,Y 456.179,Z 681,A -85,B 0,C 180,E1 -16028.166,E2 -16028.166} C_VEL
LIN {X 0,Y 456.614,Z 672.053,A -85,B 0,C 180,E1 -16029.715,E2 -16029.715} C_VEL
LIN {X 0,Y 457.095,Z 663.388,A -85,B 0,C 180,E1 -16030.948,E2 -16030.948} C_VEL
LIN {X 0,Y 457.725,Z 652.306,A -85,B 0,C 180,E1 -16032.259,E2 -16032.259} C_VEL
LIN {X 0,Y 458.328,Z 640.925,A -85,B 0,C 180,E1 -16033.365,E2 -16033.365} C_VEL
LIN {X 0,Y 459.058,Z 628.519,A -85,B 0,C 180,E1 -16034.356,E2 -16034.356} C_VEL
LIN {X 0,Y 459.841,Z 614.893,A -85,B 0,C 180,E1 -16035.234,E2 -16035.234} C_VEL
LIN {X 0,Y 460.329,Z 601.842,A -85,B 0,C 180,E1 -16035.896,E2 -16035.896} C_VEL
LIN {X 0,Y 460.903,Z 587.37,A -85,B 0,C 180,E1 -16036.443,E2 -16036.443} C_VEL
LIN {X 0,Y 461.352,Z 571.846,A -85,B 0,C 180,E1 -16036.839,E2 -16036.839} C_VEL
LIN {X 0,Y 463.651,Z 468.508,A -85,B 0,C 180,E1 -16038.949,E2 -16038.949} C_VEL
LIN {X 0,Y 460.769,Z 439.513,A -85,B 0,C 180,E1 -16039.661,E2 -16039.661} C_VEL
LIN {X 0,Y 462.309,Z 410.056,A -85,B 0,C 180,E1 -16043.199,E2 -16043.199} C_VEL
LIN {X 0,Y 463.754,Z 384.963,A -85,B 0,C 180,E1 -16046.218,E2 -16046.218} C_VEL
LIN {X 0,Y 464.442,Z 372.316,A -85,B 0,C 180,E1 -16047.747,E2 -16047.747} C_VEL
LIN {X 0,Y 461.945,Z 359.806,A -85,B 0,C 180,E1 -16049.4,E2 -16049.4} C_VEL
LIN {X 0,Y 457.643,Z 341.036,A -85,B 0,C 180,E1 -16051.938,E2 -16051.938} C_VEL
LIN {X 0,Y 457.617,Z 341.036,A -85,B 0,C 180,E1 -16054.495,E2 -16054.495} C_VEL
LIN {X 0,Y 457.556,Z 341.045,A -85,B 0,C 180,E1 -16057.759,E2 -16057.759} C_VEL
LIN {X 0,Y 457.64,Z 341.033,A -85,B 0,C 180,E1 -16060.068,E2 -16060.068} C_VEL
LIN {X 0,Y 457.605,Z 341.039,A -85,B 0,C 180,E1 -16063.536,E2 -16063.536} C_VEL
LIN {X 0,Y 457.605,Z 341.039,A -85,B 0,C 180,E1 -16066.464,E2 -16066.464} C_VEL
LIN {X 0,Y 457.651,Z 341.031,A -85,B 0,C 180,E1 -16069.998,E2 -16069.998} C_VEL
LIN {X 0,Y 457.598,Z 341.039,A -85,B 0,C 180,E1 -16073.347,E2 -16073.347} C_VEL
LIN {X 0,Y 457.62,Z 341.042,A -85,B 0,C 180,E1 -16076.563,E2 -16076.563} C_VEL
LIN {X 0,Y 457.614,Z 341.036,A -85,B 0,C 180,E1 -16079.661,E2 -16079.661} C_VEL
LIN {X 0,Y 457.641,Z 341.037,A -85,B 0,C 180,E1 -16082.667,E2 -16082.667} C_VEL
LIN {X 0,Y 457.587,Z 341.04,A -85,B 0,C 180,E1 -16085.588,E2 -16085.588} C_VEL
LIN {X 0,Y 457.661,Z 341.03,A -85,B 0,C 180,E1 -16089.004,E2 -16089.004} C_VEL
LIN {X 0,Y 457.666,Z 341.037,A -85,B 0,C 180,E1 -16092.176,E2 -16092.176} C_VEL
LIN {X 0,Y 457.696,Z 341.033,A -85,B 0,C 180,E1 -16094.879,E2 -16094.879} C_VEL
LIN {X 0,Y 465.796,Z 363.023,A -85,B 0,C 180,E1 -16095.584,E2 -16095.584} C_VEL
LIN {X 0,Y 464.766,Z 455.662,A -85,B 0,C 180,E1 -16097.018,E2 -16097.018} C_VEL
LIN {X 0,Y 464.643,Z 469.865,A -85,B 0,C 180,E1 -16097.346,E2 -16097.346} C_VEL
LIN {X 0,Y 464.326,Z 484.236,A -85,B 0,C 180,E1 -16097.863,E2 -16097.863} C_VEL
LIN {X 0,Y 463.781,Z 496.456,A -85,B 0,C 180,E1 -16098.456,E2 -16098.456} C_VEL
LIN {X 0,Y 463.141,Z 508.632,A -85,B 0,C 180,E1 -16099.213,E2 -16099.213} C_VEL
LIN {X 0,Y 462.564,Z 519.691,A -85,B 0,C 180,E1 -16100.067,E2 -16100.067} C_VEL
LIN {X 0,Y 461.676,Z 531.379,A -85,B 0,C 180,E1 -16101.164,E2 -16101.164} C_VEL
LIN {X 0,Y 460.752,Z 541.809,A -85,B 0,C 180,E1 -16102.356,E2 -16102.356} C_VEL
LIN {X 0,Y 459.783,Z 551.236,A -85,B 0,C 180,E1 -16103.659,E2 -16103.659} C_VEL
LIN {X 0,Y 459.155,Z 559.026,A -85,B 0,C 180,E1 -16104.968,E2 -16104.968} C_VEL
LIN {X 0,Y 458.327,Z 566.539,A -85,B 0,C 180,E1 -16106.495,E2 -16106.495} C_VEL
LIN {X 0,Y 457.869,Z 571.758,A -85,B 0,C 180,E1 -16107.808,E2 -16107.808} C_VEL
LIN {X 0,Y 457.35,Z 577.272,A -85,B 0,C 180,E1 -16109.561,E2 -16109.561} C_VEL
LIN {X 0,Y 457.167,Z 580.383,A -85,B 0,C 180,E1 -16110.878,E2 -16110.878} C_VEL
LIN {X 0,Y 457.106,Z 583.3,A -85,B 0,C 180,E1 -16112.635,E2 -16112.635} C_VEL
LIN {X 0,Y 456.962,Z 584.921,A -85,B 0,C 180,E1 -16114.396,E2 -16114.396} C_VEL
LIN {X 0,Y 457.071,Z 585.234,A -85,B 0,C 180,E1 -16115.962,E2 -16115.962} C_VEL
LIN {X 0,Y 456.495,Z 585.175,A -85,B 0,C 180,E1 -16116.699,E2 -16116.699} C_VEL
LIN {X 0,Y 453.775,Z 584.702,A -85,B 0,C 180,E1 -16117.897,E2 -16117.897} C_VEL
LIN {X 0,Y 451.504,Z 583.967,A -85,B 0,C 180,E1 -16118.858,E2 -16118.858} C_VEL
LIN {X 0,Y 450.62,Z 583.051,A -85,B 0,C 180,E1 -16119.595,E2 -16119.595} C_VEL
LIN {X 0,Y 450.599,Z 582.676,A -85,B 0,C 180,E1 -16119.843,E2 -16119.843} C_VEL
LIN {X 0,Y 451.345,Z 578.939,A -85,B 0,C 180,E1 -16121.639,E2 -16121.639} C_VEL
LIN {X 0,Y 452.092,Z 573.663,A -85,B 0,C 180,E1 -16123.439,E2 -16123.439} C_VEL
LIN {X 0,Y 452.872,Z 568.611,A -85,B 0,C 180,E1 -16124.786,E2 -16124.786} C_VEL
LIN {X 0,Y 453.921,Z 561.343,A -85,B 0,C 180,E1 -16126.353,E2 -16126.353} C_VEL
LIN {X 0,Y 454.981,Z 553.668,A -85,B 0,C 180,E1 -16127.701,E2 -16127.701} C_VEL
LIN {X 0,Y 456.172,Z 544.417,A -85,B 0,C 180,E1 -16129.044,E2 -16129.044} C_VEL
LIN {X 0,Y 457.319,Z 534.131,A -85,B 0,C 180,E1 -16130.276,E2 -16130.276} C_VEL
LIN {X 0,Y 458.391,Z 523.365,A -85,B 0,C 180,E1 -16131.34,E2 -16131.34} C_VEL
LIN {X 0,Y 459.484,Z 511.64,A -85,B 0,C 180,E1 -16132.284,E2 -16132.284} C_VEL
LIN {X 0,Y 460.373,Z 499.64,A -85,B 0,C 180,E1 -16133.065,E2 -16133.065} C_VEL
LIN {X 0,Y 460.819,Z 488.959,A -85,B 0,C 180,E1 -16133.635,E2 -16133.635} C_VEL
LIN {X 0,Y 461.324,Z 475.282,A -85,B 0,C 180,E1 -16134.183,E2 -16134.183} C_VEL
LIN {X 0,Y 461.617,Z 461.547,A -85,B 0,C 180,E1 -16134.556,E2 -16134.556} C_VEL
LIN {X 0,Y 462.569,Z 402.198,A -85,B 0,C 180,E1 -16135.504,E2 -16135.504} C_VEL
LIN {X 0,Y 463.059,Z 370.377,A -85,B 0,C 180,E1 -16136.005,E2 -16136.005} C_VEL
LIN {X 0,Y 452.651,Z 347.075,A -85,B 0,C 180,E1 -16136.984,E2 -16136.984} C_VEL
LIN {X 0,Y 450.712,Z 342.674,A -85,B 0,C 180,E1 -16137.173,E2 -16137.173} C_VEL
LIN {X 0,Y 450.56,Z 341.924,A -85,B 0,C 180,E1 -16137.203,E2 -16137.203} C_VEL
LIN {X 0,Y 450.544,Z 341.923,A -85,B 0,C 180,E1 -16139.835,E2 -16139.835} C_VEL
LIN {X 0,Y 450.498,Z 341.926,A -85,B 0,C 180,E1 -16142.969,E2 -16142.969} C_VEL
LIN {X 0,Y 450.485,Z 341.929,A -85,B 0,C 180,E1 -16146.218,E2 -16146.218} C_VEL
LIN {X 0,Y 450.528,Z 341.922,A -85,B 0,C 180,E1 -16148.98,E2 -16148.98} C_VEL
LIN {X 0,Y 450.528,Z 341.925,A -85,B 0,C 180,E1 -16151.954,E2 -16151.954} C_VEL
LIN {X 0,Y 450.558,Z 341.917,A -85,B 0,C 180,E1 -16154.393,E2 -16154.393} C_VEL
LIN {X 0,Y 450.55,Z 341.918,A -85,B 0,C 180,E1 -16156.944,E2 -16156.944} C_VEL
LIN {X 0,Y 450.513,Z 341.925,A -85,B 0,C 180,E1 -16159.627,E2 -16159.627} C_VEL
LIN {X 0,Y 450.481,Z 341.898,A -85,B 0,C 180,E1 -16162.67,E2 -16162.67} C_VEL
LIN {X 0,Y 450.529,Z 341.915,A -85,B 0,C 180,E1 -16165.965,E2 -16165.965} C_VEL
LIN {X 0,Y 450.521,Z 341.915,A -85,B 0,C 180,E1 -16169.131,E2 -16169.131} C_VEL
LIN {X 0,Y 450.551,Z 341.916,A -85,B 0,C 180,E1 -16171.188,E2 -16171.188} C_VEL
LIN {X 0,Y 450.548,Z 341.912,A -85,B 0,C 180,E1 -16174.383,E2 -16174.383} C_VEL
LIN {X 0,Y 450.518,Z 341.923,A -85,B 0,C 180,E1 -16177.127,E2 -16177.127} C_VEL
LIN {X 0,Y 450.583,Z 341.919,A -85,B 0,C 180,E1 -16179.905,E2 -16179.905} C_VEL
LIN {X 0,Y 456.367,Z 362.195,A -85,B 0,C 180,E1 -16180.5,E2 -16180.5} C_VEL
LIN {X 0,Y 454.375,Z 460.18,A -85,B 0,C 180,E1 -16182.535,E2 -16182.535} C_VEL
LIN {X 0,Y 454.163,Z 475.632,A -85,B 0,C 180,E1 -16183.044,E2 -16183.044} C_VEL
LIN {X 0,Y 453.764,Z 490.023,A -85,B 0,C 180,E1 -16183.7,E2 -16183.7} C_VEL
LIN {X 0,Y 453.194,Z 504.049,A -85,B 0,C 180,E1 -16184.537,E2 -16184.537} C_VEL
LIN {X 0,Y 452.634,Z 517.541,A -85,B 0,C 180,E1 -16185.55,E2 -16185.55} C_VEL
LIN {X 0,Y 451.995,Z 529.732,A -85,B 0,C 180,E1 -16186.672,E2 -16186.672} C_VEL
LIN {X 0,Y 451.575,Z 540.657,A -85,B 0,C 180,E1 -16187.901,E2 -16187.901} C_VEL
LIN {X 0,Y 451.051,Z 550.71,A -85,B 0,C 180,E1 -16189.26,E2 -16189.26} C_VEL
LIN {X 0,Y 450.573,Z 559.001,A -85,B 0,C 180,E1 -16190.605,E2 -16190.605} C_VEL
LIN {X 0,Y 450.208,Z 566.962,A -85,B 0,C 180,E1 -16192.176,E2 -16192.176} C_VEL
LIN {X 0,Y 449.991,Z 573.3,A -85,B 0,C 180,E1 -16193.744,E2 -16193.744} C_VEL
LIN {X 0,Y 449.854,Z 578.844,A -85,B 0,C 180,E1 -16195.535,E2 -16195.535} C_VEL
LIN {X 0,Y 449.884,Z 582.808,A -85,B 0,C 180,E1 -16197.323,E2 -16197.323} C_VEL
LIN {X 0,Y 449.935,Z 585.285,A -85,B 0,C 180,E1 -16199.108,E2 -16199.108} C_VEL
LIN {X 0,Y 450.171,Z 586.276,A -85,B 0,C 180,E1 -16200.891,E2 -16200.891} C_VEL
LIN {X 0,Y 450.552,Z 585.843,A -85,B 0,C 180,E1 -16202.673,E2 -16202.673} C_VEL
LIN {X 0,Y 451.272,Z 583.956,A -85,B 0,C 180,E1 -16204.451,E2 -16204.451} C_VEL
LIN {X 0,Y 452.026,Z 580.621,A -85,B 0,C 180,E1 -16206.227,E2 -16206.227} C_VEL
LIN {X 0,Y 452.744,Z 577.051,A -85,B 0,C 180,E1 -16207.556,E2 -16207.556} C_VEL
LIN {X 0,Y 453.848,Z 572.105,A -85,B 0,C 180,E1 -16208.978,E2 -16208.978} C_VEL
LIN {X 0,Y 455.092,Z 564.819,A -85,B 0,C 180,E1 -16210.643,E2 -16210.643} C_VEL
LIN {X 0,Y 456.473,Z 556.251,A -85,B 0,C 180,E1 -16212.18,E2 -16212.18} C_VEL
LIN {X 0,Y 457.79,Z 547.276,A -85,B 0,C 180,E1 -16213.493,E2 -16213.493} C_VEL
LIN {X 0,Y 458.867,Z 538.41,A -85,B 0,C 180,E1 -16214.588,E2 -16214.588} C_VEL
LIN {X 0,Y 460.346,Z 526.611,A -85,B 0,C 180,E1 -16215.782,E2 -16215.782} C_VEL
LIN {X 0,Y 461.684,Z 514.717,A -85,B 0,C 180,E1 -16216.754,E2 -16216.754} C_VEL
LIN {X 0,Y 462.804,Z 501.753,A -85,B 0,C 180,E1 -16217.619,E2 -16217.619} C_VEL
LIN {X 0,Y 463.632,Z 488.472,A -85,B 0,C 180,E1 -16218.326,E2 -16218.326} C_VEL
LIN {X 0,Y 464.239,Z 475.056,A -85,B 0,C 180,E1 -16218.871,E2 -16218.871} C_VEL
LIN {X 0,Y 464.688,Z 458.728,A -85,B 0,C 180,E1 -16219.338,E2 -16219.338} C_VEL
LIN {X 0,Y 468.613,Z 385.57,A -85,B 0,C 180,E1 -16221.086,E2 -16221.086} C_VEL
LIN {X 0,Y 469.142,Z 375.66,A -85,B 0,C 180,E1 -16221.332,E2 -16221.332} C_VEL
LIN {X 0,Y 463.157,Z 363.545,A -85,B 0,C 180,E1 -16222.302,E2 -16222.302} C_VEL
LIN {X 0,Y 457.268,Z 353.511,A -85,B 0,C 180,E1 -16223.269,E2 -16223.269} C_VEL
LIN {X 0,Y 455.115,Z 350.053,A -85,B 0,C 180,E1 -16223.646,E2 -16223.646} C_VEL
LIN {X 0,Y 452.802,Z 346.246,A -85,B 0,C 180,E1 -16224.061,E2 -16224.061} C_VEL
LIN {X 0,Y 451.155,Z 343.988,A -85,B 0,C 180,E1 -16224.343,E2 -16224.343} C_VEL
LIN {X 0,Y 450.562,Z 341.923,A -85,B 0,C 180,E1 -16224.515,E2 -16224.515} C_VEL
LIN {X 0,Y 450.582,Z 341.918,A -85,B 0,C 180,E1 -16227.798,E2 -16227.798} C_VEL
LIN {X 0,Y 450.571,Z 341.917,A -85,B 0,C 180,E1 -16230.864,E2 -16230.864} C_VEL
LIN {X 0,Y 450.569,Z 341.914,A -85,B 0,C 180,E1 -16234.031,E2 -16234.031} C_VEL
LIN {X 0,Y 450.521,Z 341.916,A -85,B 0,C 180,E1 -16237.326,E2 -16237.326} C_VEL
LIN {X 0,Y 450.53,Z 341.913,A -85,B 0,C 180,E1 -16240.376,E2 -16240.376} C_VEL
LIN {X 0,Y 450.542,Z 341.919,A -85,B 0,C 180,E1 -16243.161,E2 -16243.161} C_VEL
LIN {X 0,Y 450.556,Z 341.915,A -85,B 0,C 180,E1 -16245.653,E2 -16245.653} C_VEL
LIN {X 0,Y 450.538,Z 341.919,A -85,B 0,C 180,E1 -16248.266,E2 -16248.266} C_VEL
LIN {X 0,Y 450.493,Z 341.925,A -85,B 0,C 180,E1 -16251.542,E2 -16251.542} C_VEL
LIN {X 0,Y 450.471,Z 341.923,A -85,B 0,C 180,E1 -16254.878,E2 -16254.878} C_VEL
LIN {X 0,Y 450.534,Z 342.037,A -85,B 0,C 180,E1 -16256.502,E2 -16256.502} C_VEL
LIN {X 0,Y 454.014,Z 355.812,A -85,B 0,C 180,E1 -16258.88,E2 -16258.88} C_VEL
LIN {X 0,Y 457.229,Z 370.33,A -85,B 0,C 180,E1 -16261.266,E2 -16261.266} C_VEL
LIN {X 0,Y 457.74,Z 374.609,A -85,B 0,C 180,E1 -16261.93,E2 -16261.93} C_VEL
LIN {X 0,Y 455.455,Z 397.967,A -85,B 0,C 180,E1 -16265.241,E2 -16265.241} C_VEL
LIN {X 0,Y 460.051,Z 426.653,A -85,B 0,C 180,E1 -16266.631,E2 -16266.631} C_VEL
LIN {X 0,Y 462.726,Z 448.985,A -85,B 0,C 180,E1 -16267.547,E2 -16267.547} C_VEL
LIN {X 0,Y 464.28,Z 474.734,A -85,B 0,C 180,E1 -16268.43,E2 -16268.43} C_VEL
LIN {X 0,Y 460.2,Z 555.543,A -85,B 0,C 180,E1 -16270.35,E2 -16270.35} C_VEL
LIN {X 0,Y 458.928,Z 571.354,A -85,B 0,C 180,E1 -16270.901,E2 -16270.901} C_VEL
LIN {X 0,Y 457.721,Z 585.988,A -85,B 0,C 180,E1 -16271.5,E2 -16271.5} C_VEL
LIN {X 0,Y 456.369,Z 599.476,A -85,B 0,C 180,E1 -16272.239,E2 -16272.239} C_VEL
LIN {X 0,Y 454.972,Z 611.853,A -85,B 0,C 180,E1 -16273.107,E2 -16273.107} C_VEL
LIN {X 0,Y 453.543,Z 624.393,A -85,B 0,C 180,E1 -16274.205,E2 -16274.205} C_VEL
LIN {X 0,Y 452.134,Z 635.618,A -85,B 0,C 180,E1 -16275.419,E2 -16275.419} C_VEL
LIN {X 0,Y 451.054,Z 645.739,A -85,B 0,C 180,E1 -16276.758,E2 -16276.758} C_VEL
LIN {X 0,Y 450.664,Z 650.411,A -85,B 0,C 180,E1 -16277.432,E2 -16277.432} C_VEL
LIN {X 0,Y 449.984,Z 661.918,A -85,B 0,C 180,E1 -16278.712,E2 -16278.712} C_VEL
LIN {X 0,Y 449.559,Z 670.824,A -85,B 0,C 180,E1 -16279.905,E2 -16279.905} C_VEL
LIN {X 0,Y 449.178,Z 679.244,A -85,B 0,C 180,E1 -16281.255,E2 -16281.255} C_VEL
LIN {X 0,Y 448.892,Z 687.264,A -85,B 0,C 180,E1 -16282.829,E2 -16282.829} C_VEL
LIN {X 0,Y 448.741,Z 692.787,A -85,B 0,C 180,E1 -16284.177,E2 -16284.177} C_VEL
LIN {X 0,Y 448.644,Z 697.242,A -85,B 0,C 180,E1 -16285.523,E2 -16285.523} C_VEL
LIN {X 0,Y 448.592,Z 701.68,A -85,B 0,C 180,E1 -16287.315,E2 -16287.315} C_VEL
LIN {X 0,Y 448.582,Z 704.534,A -85,B 0,C 180,E1 -16289.105,E2 -16289.105} C_VEL
LIN {X 0,Y 448.552,Z 705.842,A -85,B 0,C 180,E1 -16290.895,E2 -16290.895} C_VEL
LIN {X 0,Y 448.594,Z 705.661,A -85,B 0,C 180,E1 -16292.685,E2 -16292.685} C_VEL
LIN {X 0,Y 448.712,Z 704.019,A -85,B 0,C 180,E1 -16294.476,E2 -16294.476} C_VEL
LIN {X 0,Y 449.044,Z 700.897,A -85,B 0,C 180,E1 -16296.269,E2 -16296.269} C_VEL
LIN {X 0,Y 449.547,Z 696.233,A -85,B 0,C 180,E1 -16298.061,E2 -16298.061} C_VEL
LIN {X 0,Y 450.085,Z 691.58,A -85,B 0,C 180,E1 -16299.405,E2 -16299.405} C_VEL
LIN {X 0,Y 451.093,Z 684.867,A -85,B 0,C 180,E1 -16300.965,E2 -16300.965} C_VEL
LIN {X 0,Y 452.156,Z 676.14,A -85,B 0,C 180,E1 -16302.592,E2 -16302.592} C_VEL
LIN {X 0,Y 453.566,Z 666.196,A -85,B 0,C 180,E1 -16304.077,E2 -16304.077} C_VEL
LIN {X 0,Y 455.065,Z 655.398,A -85,B 0,C 180,E1 -16305.397,E2 -16305.397} C_VEL
LIN {X 0,Y 456.425,Z 644.583,A -85,B 0,C 180,E1 -16306.493,E2 -16306.493} C_VEL
LIN {X 0,Y 457.885,Z 632.923,A -85,B 0,C 180,E1 -16307.47,E2 -16307.47} C_VEL
LIN {X 0,Y 459.262,Z 620.25,A -85,B 0,C 180,E1 -16308.334,E2 -16308.334} C_VEL
LIN {X 0,Y 460.652,Z 606.318,A -85,B 0,C 180,E1 -16309.082,E2 -16309.082} C_VEL
LIN {X 0,Y 461.717,Z 593.826,A -85,B 0,C 180,E1 -16309.601,E2 -16309.601} C_VEL
LIN {X 0,Y 462.739,Z 578.742,A -85,B 0,C 180,E1 -16310.053,E2 -16310.053} C_VEL
LIN {X 0,Y 467.762,Z 489.682,A -85,B 0,C 180,E1 -16312.221,E2 -16312.221} C_VEL
LIN {X 0,Y 468.493,Z 474.921,A -85,B 0,C 180,E1 -16312.61,E2 -16312.61} C_VEL
LIN {X 0,Y 467.8,Z 458.953,A -85,B 0,C 180,E1 -16313.181,E2 -16313.181} C_VEL
LIN {X 0,Y 465.694,Z 437.926,A -85,B 0,C 180,E1 -16314.082,E2 -16314.082} C_VEL
LIN {X 0,Y 465.103,Z 423.358,A -85,B 0,C 180,E1 -16315.068,E2 -16315.068} C_VEL
LIN {X 0,Y 464.645,Z 404.973,A -85,B 0,C 180,E1 -16316.49,E2 -16316.49} C_VEL
LIN {X 0,Y 464.388,Z 385.643,A -85,B 0,C 180,E1 -16318.218,E2 -16318.218} C_VEL
LIN {X 0,Y 464.268,Z 377.693,A -85,B 0,C 180,E1 -16319.024,E2 -16319.024} C_VEL
LIN {X 0,Y 462.96,Z 368.872,A -85,B 0,C 180,E1 -16320.259,E2 -16320.259} C_VEL
LIN {X 0,Y 461.936,Z 362.061,A -85,B 0,C 180,E1 -16321.354,E2 -16321.354} C_VEL
LIN {X 0,Y 461.325,Z 360.19,A -85,B 0,C 180,E1 -16321.759,E2 -16321.759} C_VEL
LIN {X 0,Y 459.072,Z 356.299,A -85,B 0,C 180,E1 -16322.946,E2 -16322.946} C_VEL
LIN {X 0,Y 456.492,Z 351.932,A -85,B 0,C 180,E1 -16324.592,E2 -16324.592} C_VEL
LIN {X 0,Y 454.672,Z 349.758,A -85,B 0,C 180,E1 -16325.832,E2 -16325.832} C_VEL
LIN {X 0,Y 453.76,Z 347.387,A -85,B 0,C 180,E1 -16327.015,E2 -16327.015} C_VEL
LIN {X 0,Y 452.002,Z 345.495,A -85,B 0,C 180,E1 -16329.211,E2 -16329.211} C_VEL
LIN {X 0,Y 451.529,Z 344.809,A -85,B 0,C 180,E1 -16330.657,E2 -16330.657} C_VEL
LIN {X 0,Y 451.478,Z 344.686,A -85,B 0,C 180,E1 -16331.867,E2 -16331.867} C_VEL
LIN {X 0,Y 452.136,Z 345.598,A -85,B 0,C 180,E1 -16334.198,E2 -16334.198} C_VEL
LIN {X 0,Y 453.393,Z 347.053,A -85,B 0,C 180,E1 -16335.957,E2 -16335.957} C_VEL
LIN {X 0,Y 454.57,Z 350.017,A -85,B 0,C 180,E1 -16337.7,E2 -16337.7} C_VEL
LIN {X 0,Y 455.795,Z 352.182,A -85,B 0,C 180,E1 -16338.852,E2 -16338.852} C_VEL
LIN {X 0,Y 457.722,Z 356.18,A -85,B 0,C 180,E1 -16340.529,E2 -16340.529} C_VEL
LIN {X 0,Y 460.205,Z 361.971,A -85,B 0,C 180,E1 -16342.497,E2 -16342.497} C_VEL
LIN {X 0,Y 462.806,Z 368.625,A -85,B 0,C 180,E1 -16344.379,E2 -16344.379} C_VEL
LIN {X 0,Y 465.16,Z 375.911,A -85,B 0,C 180,E1 -16346.141,E2 -16346.141} C_VEL
LIN {X 0,Y 467.604,Z 385.106,A -85,B 0,C 180,E1 -16348.062,E2 -16348.062} C_VEL
LIN {X 0,Y 469.097,Z 392.849,A -85,B 0,C 180,E1 -16349.491,E2 -16349.491} C_VEL
LIN {X 0,Y 469.205,Z 394.612,A -85,B 0,C 180,E1 -16349.775,E2 -16349.775} C_VEL
LIN {X 0,Y 466.182,Z 417.055,A -85,B 0,C 180,E1 -16352.732,E2 -16352.732} C_VEL
LIN {X 0,Y 463.49,Z 439.906,A -85,B 0,C 180,E1 -16355.668,E2 -16355.668} C_VEL
LIN {X 0,Y 466.911,Z 458.251,A -85,B 0,C 180,E1 -16356.62,E2 -16356.62} C_VEL
LIN {X 0,Y 468.843,Z 472.418,A -85,B 0,C 180,E1 -16357.25,E2 -16357.25} C_VEL
LIN {X 0,Y 468.987,Z 475.791,A -85,B 0,C 180,E1 -16357.367,E2 -16357.367} C_VEL
LIN {X 0,Y 464.366,Z 556.678,A -85,B 0,C 180,E1 -16359.337,E2 -16359.337} C_VEL
LIN {X 0,Y 462.839,Z 583.774,A -85,B 0,C 180,E1 -16360.004,E2 -16360.004} C_VEL
LIN {X 0,Y 461.696,Z 597.626,A -85,B 0,C 180,E1 -16360.503,E2 -16360.503} C_VEL
LIN {X 0,Y 460.219,Z 612.807,A -85,B 0,C 180,E1 -16361.245,E2 -16361.245} C_VEL
LIN {X 0,Y 458.838,Z 626.373,A -85,B 0,C 180,E1 -16362.108,E2 -16362.108} C_VEL
LIN {X 0,Y 457.145,Z 639.924,A -85,B 0,C 180,E1 -16363.19,E2 -16363.19} C_VEL
LIN {X 0,Y 455.555,Z 652.129,A -85,B 0,C 180,E1 -16364.391,E2 -16364.391} C_VEL
LIN {X 0,Y 454.295,Z 661.392,A -85,B 0,C 180,E1 -16365.49,E2 -16365.49} C_VEL
LIN {X 0,Y 452.847,Z 671.162,A -85,B 0,C 180,E1 -16366.871,E2 -16366.871} C_VEL
LIN {X 0,Y 451.784,Z 679.791,A -85,B 0,C 180,E1 -16368.372,E2 -16368.372} C_VEL
LIN {X 0,Y 450.778,Z 686.169,A -85,B 0,C 180,E1 -16369.707,E2 -16369.707} C_VEL
LIN {X 0,Y 449.836,Z 692.917,A -85,B 0,C 180,E1 -16371.493,E2 -16371.493} C_VEL
LIN {X 0,Y 449.196,Z 697.979,A -85,B 0,C 180,E1 -16373.284,E2 -16373.284} C_VEL
LIN {X 0,Y 448.832,Z 700.728,A -85,B 0,C 180,E1 -16374.627,E2 -16374.627} C_VEL
LIN {X 0,Y 448.592,Z 703.089,A -85,B 0,C 180,E1 -16376.419,E2 -16376.419} C_VEL
LIN {X 0,Y 448.504,Z 704.002,A -85,B 0,C 180,E1 -16378.21,E2 -16378.21} C_VEL
LIN {X 0,Y 448.485,Z 703.466,A -85,B 0,C 180,E1 -16380,E2 -16380} C_VEL
LIN {X 0,Y 448.504,Z 701.44,A -85,B 0,C 180,E1 -16381.79,E2 -16381.79} C_VEL
LIN {X 0,Y 448.545,Z 697.871,A -85,B 0,C 180,E1 -16383.581,E2 -16383.581} C_VEL
LIN {X 0,Y 448.654,Z 692.689,A -85,B 0,C 180,E1 -16385.375,E2 -16385.375} C_VEL
LIN {X 0,Y 448.822,Z 687.62,A -85,B 0,C 180,E1 -16386.722,E2 -16386.722} C_VEL
LIN {X 0,Y 449.119,Z 680.281,A -85,B 0,C 180,E1 -16388.295,E2 -16388.295} C_VEL
LIN {X 0,Y 449.519,Z 672.571,A -85,B 0,C 180,E1 -16389.643,E2 -16389.643} C_VEL
LIN {X 0,Y 449.999,Z 663.427,A -85,B 0,C 180,E1 -16390.973,E2 -16390.973} C_VEL
LIN {X 0,Y 450.612,Z 653.054,A -85,B 0,C 180,E1 -16392.228,E2 -16392.228} C_VEL
LIN {X 0,Y 451.212,Z 641.816,A -85,B 0,C 180,E1 -16393.351,E2 -16393.351} C_VEL
LIN {X 0,Y 451.941,Z 629.579,A -85,B 0,C 180,E1 -16394.358,E2 -16394.358} C_VEL
LIN {X 0,Y 452.738,Z 616.19,A -85,B 0,C 180,E1 -16395.249,E2 -16395.249} C_VEL
LIN {X 0,Y 453.231,Z 603.482,A -85,B 0,C 180,E1 -16395.922,E2 -16395.922} C_VEL
LIN {X 0,Y 453.766,Z 588.957,A -85,B 0,C 180,E1 -16396.507,E2 -16396.507} C_VEL
LIN {X 0,Y 454.274,Z 573.779,A -85,B 0,C 180,E1 -16396.92,E2 -16396.92} C_VEL
LIN {X 0,Y 456.674,Z 468.519,A -85,B 0,C 180,E1 -16399.13,E2 -16399.13} C_VEL
LIN {X 0,Y 453.768,Z 439.564,A -85,B 0,C 180,E1 -16399.853,E2 -16399.853} C_VEL
LIN {X 0,Y 455.362,Z 410.828,A -85,B 0,C 180,E1 -16403.334,E2 -16403.334} C_VEL
LIN {X 0,Y 456.83,Z 385.596,A -85,B 0,C 180,E1 -16406.401,E2 -16406.401} C_VEL
LIN {X 0,Y 457.465,Z 372.815,A -85,B 0,C 180,E1 -16407.964,E2 -16407.964} C_VEL
LIN {X 0,Y 453.304,Z 353.782,A -85,B 0,C 180,E1 -16410.512,E2 -16410.512} C_VEL
LIN {X 0,Y 450.596,Z 341.914,A -85,B 0,C 180,E1 -16412.169,E2 -16412.169} C_VEL
LIN {X 0,Y 450.578,Z 341.918,A -85,B 0,C 180,E1 -16415.113,E2 -16415.113} C_VEL
LIN {X 0,Y 450.549,Z 341.917,A -85,B 0,C 180,E1 -16418.452,E2 -16418.452} C_VEL
LIN {X 0,Y 450.553,Z 341.919,A -85,B 0,C 180,E1 -16420.765,E2 -16420.765} C_VEL
LIN {X 0,Y 450.574,Z 341.919,A -85,B 0,C 180,E1 -16423.158,E2 -16423.158} C_VEL
LIN {X 0,Y 450.58,Z 341.913,A -85,B 0,C 180,E1 -16425.651,E2 -16425.651} C_VEL
LIN {X 0,Y 450.552,Z 341.917,A -85,B 0,C 180,E1 -16428.265,E2 -16428.265} C_VEL
LIN {X 0,Y 450.565,Z 341.919,A -85,B 0,C 180,E1 -16431.014,E2 -16431.014} C_VEL
LIN {X 0,Y 450.556,Z 341.915,A -85,B 0,C 180,E1 -16433.941,E2 -16433.941} C_VEL
LIN {X 0,Y 450.574,Z 341.915,A -85,B 0,C 180,E1 -16437.084,E2 -16437.084} C_VEL
LIN {X 0,Y 450.582,Z 341.919,A -85,B 0,C 180,E1 -16440.522,E2 -16440.522} C_VEL
LIN {X 0,Y 450.588,Z 341.912,A -85,B 0,C 180,E1 -16443.204,E2 -16443.204} C_VEL
LIN {X 0,Y 450.584,Z 341.917,A -85,B 0,C 180,E1 -16446.517,E2 -16446.517} C_VEL
LIN {X 0,Y 450.598,Z 341.915,A -85,B 0,C 180,E1 -16450.002,E2 -16450.002} C_VEL
LIN {X 0,Y 450.598,Z 341.911,A -85,B 0,C 180,E1 -16452.822,E2 -16452.822} C_VEL
LIN {X 0,Y 450.642,Z 341.911,A -85,B 0,C 180,E1 -16454.592,E2 -16454.592} C_VEL
LIN {X 0,Y 459.16,Z 364.849,A -85,B 0,C 180,E1 -16455.34,E2 -16455.34} C_VEL
LIN {X 0,Y 457.995,Z 451.229,A -85,B 0,C 180,E1 -16456.687,E2 -16456.687} C_VEL
LIN {X 0,Y 457.944,Z 467.483,A -85,B 0,C 180,E1 -16457.018,E2 -16457.018} C_VEL
LIN {X 0,Y 457.641,Z 480.898,A -85,B 0,C 180,E1 -16457.459,E2 -16457.459} C_VEL
LIN {X 0,Y 457.142,Z 494.124,A -85,B 0,C 180,E1 -16458.062,E2 -16458.062} C_VEL
LIN {X 0,Y 456.458,Z 506.96,A -85,B 0,C 180,E1 -16458.829,E2 -16458.829} C_VEL
LIN {X 0,Y 455.778,Z 519.466,A -85,B 0,C 180,E1 -16459.782,E2 -16459.782} C_VEL
LIN {X 0,Y 454.847,Z 531.546,A -85,B 0,C 180,E1 -16460.918,E2 -16460.918} C_VEL
LIN {X 0,Y 453.939,Z 541.207,A -85,B 0,C 180,E1 -16462.017,E2 -16462.017} C_VEL
LIN {X 0,Y 452.963,Z 550.856,A -85,B 0,C 180,E1 -16463.34,E2 -16463.34} C_VEL
LIN {X 0,Y 452.193,Z 558.858,A -85,B 0,C 180,E1 -16464.667,E2 -16464.667} C_VEL
LIN {X 0,Y 451.514,Z 565.542,A -85,B 0,C 180,E1 -16465.997,E2 -16465.997} C_VEL
LIN {X 0,Y 450.952,Z 571.113,A -85,B 0,C 180,E1 -16467.329,E2 -16467.329} C_VEL
LIN {X 0,Y 450.431,Z 576.951,A -85,B 0,C 180,E1 -16469.109,E2 -16469.109} C_VEL
LIN {X 0,Y 450.114,Z 581.245,A -85,B 0,C 180,E1 -16470.892,E2 -16470.892} C_VEL
LIN {X 0,Y 450.048,Z 584.128,A -85,B 0,C 180,E1 -16472.676,E2 -16472.676} C_VEL
LIN {X 0,Y 449.91,Z 585.715,A -85,B 0,C 180,E1 -16474.465,E2 -16474.465} C_VEL
LIN {X 0,Y 450.072,Z 585.992,A -85,B 0,C 180,E1 -16476.254,E2 -16476.254} C_VEL
LIN {X 0,Y 450.274,Z 584.989,A -85,B 0,C 180,E1 -16478.048,E2 -16478.048} C_VEL
LIN {X 0,Y 450.599,Z 582.676,A -85,B 0,C 180,E1 -16479.843,E2 -16479.843} C_VEL
LIN {X 0,Y 450.153,Z 581.533,A -85,B 0,C 180,E1 -16480.579,E2 -16480.579} C_VEL
LIN {X 0,Y 447.746,Z 579.323,A -85,B 0,C 180,E1 -16481.777,E2 -16481.777} C_VEL
LIN {X 0,Y 445.448,Z 576.428,A -85,B 0,C 180,E1 -16482.961,E2 -16482.961} C_VEL
LIN {X 0,Y 445.176,Z 574.212,A -85,B 0,C 180,E1 -16483.666,E2 -16483.666} C_VEL
LIN {X 0,Y 446.008,Z 569.183,A -85,B 0,C 180,E1 -16485.019,E2 -16485.019} C_VEL
LIN {X 0,Y 447.067,Z 561.945,A -85,B 0,C 180,E1 -16486.593,E2 -16486.593} C_VEL
LIN {X 0,Y 448.163,Z 554.276,A -85,B 0,C 180,E1 -16487.956,E2 -16487.956} C_VEL
LIN {X 0,Y 449.423,Z 544.808,A -85,B 0,C 180,E1 -16489.341,E2 -16489.341} C_VEL
LIN {X 0,Y 450.662,Z 534.443,A -85,B 0,C 180,E1 -16490.589,E2 -16490.589} C_VEL
LIN {X 0,Y 451.837,Z 522.804,A -85,B 0,C 180,E1 -16491.737,E2 -16491.737} C_VEL
LIN {X 0,Y 453.02,Z 510.154,A -85,B 0,C 180,E1 -16492.74,E2 -16492.74} C_VEL
LIN {X 0,Y 453.848,Z 497.566,A -85,B 0,C 180,E1 -16493.537,E2 -16493.537} C_VEL
LIN {X 0,Y 454.48,Z 483.969,A -85,B 0,C 180,E1 -16494.202,E2 -16494.202} C_VEL
LIN {X 0,Y 454.901,Z 470.05,A -85,B 0,C 180,E1 -16494.691,E2 -16494.691} C_VEL
LIN {X 0,Y 455.112,Z 454.662,A -85,B 0,C 180,E1 -16495.024,E2 -16495.024} C_VEL
LIN {X 0,Y 456.508,Z 372.04,A -85,B 0,C 180,E1 -16496.339,E2 -16496.339} C_VEL
LIN {X 0,Y 445.707,Z 348.138,A -85,B 0,C 180,E1 -16497.377,E2 -16497.377} C_VEL
LIN {X 0,Y 443.721,Z 343.856,A -85,B 0,C 180,E1 -16497.572,E2 -16497.572} C_VEL
LIN {X 0,Y 443.521,Z 342.796,A -85,B 0,C 180,E1 -16497.639,E2 -16497.639} C_VEL
LIN {X 0,Y 443.47,Z 342.805,A -85,B 0,C 180,E1 -16500.36,E2 -16500.36} C_VEL
LIN {X 0,Y 443.435,Z 342.806,A -85,B 0,C 180,E1 -16503.563,E2 -16503.563} C_VEL
LIN {X 0,Y 443.431,Z 342.807,A -85,B 0,C 180,E1 -16506.888,E2 -16506.888} C_VEL
LIN {X 0,Y 443.463,Z 342.802,A -85,B 0,C 180,E1 -16509.29,E2 -16509.29} C_VEL
LIN {X 0,Y 443.486,Z 342.801,A -85,B 0,C 180,E1 -16512.07,E2 -16512.07} C_VEL
LIN {X 0,Y 443.496,Z 342.794,A -85,B 0,C 180,E1 -16515.294,E2 -16515.294} C_VEL
LIN {X 0,Y 443.491,Z 342.798,A -85,B 0,C 180,E1 -16518.444,E2 -16518.444} C_VEL
LIN {X 0,Y 443.466,Z 342.779,A -85,B 0,C 180,E1 -16521.975,E2 -16521.975} C_VEL
LIN {X 0,Y 443.495,Z 342.783,A -85,B 0,C 180,E1 -16525.349,E2 -16525.349} C_VEL
LIN {X 0,Y 443.499,Z 342.789,A -85,B 0,C 180,E1 -16528.588,E2 -16528.588} C_VEL
LIN {X 0,Y 443.499,Z 342.8,A -85,B 0,C 180,E1 -16531.718,E2 -16531.718} C_VEL
LIN {X 0,Y 443.484,Z 342.791,A -85,B 0,C 180,E1 -16534.758,E2 -16534.758} C_VEL
LIN {X 0,Y 443.471,Z 342.799,A -85,B 0,C 180,E1 -16537.724,E2 -16537.724} C_VEL
LIN {X 0,Y 443.535,Z 342.793,A -85,B 0,C 180,E1 -16539.721,E2 -16539.721} C_VEL
LIN {X 0,Y 449.35,Z 363.283,A -85,B 0,C 180,E1 -16540.346,E2 -16540.346} C_VEL
LIN {X 0,Y 447.361,Z 461.083,A -85,B 0,C 180,E1 -16542.428,E2 -16542.428} C_VEL
LIN {X 0,Y 447.153,Z 476.468,A -85,B 0,C 180,E1 -16542.946,E2 -16542.946} C_VEL
LIN {X 0,Y 446.694,Z 490.713,A -85,B 0,C 180,E1 -16543.605,E2 -16543.605} C_VEL
LIN {X 0,Y 446.186,Z 504.017,A -85,B 0,C 180,E1 -16544.405,E2 -16544.405} C_VEL
LIN {X 0,Y 445.603,Z 517.647,A -85,B 0,C 180,E1 -16545.433,E2 -16545.433} C_VEL
LIN {X 0,Y 444.968,Z 529.961,A -85,B 0,C 180,E1 -16546.574,E2 -16546.574} C_VEL
LIN {X 0,Y 444.524,Z 541.092,A -85,B 0,C 180,E1 -16547.834,E2 -16547.834} C_VEL
LIN {X 0,Y 443.941,Z 551.886,A -85,B 0,C 180,E1 -16549.316,E2 -16549.316} C_VEL
LIN {X 0,Y 443.473,Z 560.127,A -85,B 0,C 180,E1 -16550.683,E2 -16550.683} C_VEL
LIN {X 0,Y 443.128,Z 568.039,A -85,B 0,C 180,E1 -16552.278,E2 -16552.278} C_VEL
LIN {X 0,Y 442.914,Z 573.528,A -85,B 0,C 180,E1 -16553.644,E2 -16553.644} C_VEL
LIN {X 0,Y 442.798,Z 578.724,A -85,B 0,C 180,E1 -16555.259,E2 -16555.259} C_VEL
LIN {X 0,Y 442.812,Z 581.503,A -85,B 0,C 180,E1 -16556.372,E2 -16556.372} C_VEL
LIN {X 0,Y 442.847,Z 584.852,A -85,B 0,C 180,E1 -16558.187,E2 -16558.187} C_VEL
LIN {X 0,Y 442.941,Z 586.762,A -85,B 0,C 180,E1 -16560,E2 -16560} C_VEL
LIN {X 0,Y 443.3,Z 587.18,A -85,B 0,C 180,E1 -16561.811,E2 -16561.811} C_VEL
LIN {X 0,Y 443.887,Z 586.152,A -85,B 0,C 180,E1 -16563.619,E2 -16563.619} C_VEL
LIN {X 0,Y 444.7,Z 583.68,A -85,B 0,C 180,E1 -16565.423,E2 -16565.423} C_VEL
LIN {X 0,Y 445.544,Z 579.734,A -85,B 0,C 180,E1 -16567.225,E2 -16567.225} C_VEL
LIN {X 0,Y 446.552,Z 575.626,A -85,B 0,C 180,E1 -16568.57,E2 -16568.57} C_VEL
LIN {X 0,Y 447.619,Z 570.527,A -85,B 0,C 180,E1 -16569.912,E2 -16569.912} C_VEL
LIN {X 0,Y 448.913,Z 563.206,A -85,B 0,C 180,E1 -16571.475,E2 -16571.475} C_VEL
LIN {X 0,Y 450.24,Z 555.494,A -85,B 0,C 180,E1 -16572.808,E2 -16572.808} C_VEL
LIN {X 0,Y 451.628,Z 546.174,A -85,B 0,C 180,E1 -16574.139,E2 -16574.139} C_VEL
LIN {X 0,Y 453.03,Z 535.865,A -85,B 0,C 180,E1 -16575.353,E2 -16575.353} C_VEL
LIN {X 0,Y 454.503,Z 524.506,A -85,B 0,C 180,E1 -16576.45,E2 -16576.45} C_VEL
LIN {X 0,Y 455.809,Z 512.445,A -85,B 0,C 180,E1 -16577.407,E2 -16577.407} C_VEL
LIN {X 0,Y 456.941,Z 498.99,A -85,B 0,C 180,E1 -16578.269,E2 -16578.269} C_VEL
LIN {X 0,Y 457.773,Z 484.888,A -85,B 0,C 180,E1 -16578.974,E2 -16578.974} C_VEL
LIN {X 0,Y 458.396,Z 469.816,A -85,B 0,C 180,E1 -16579.527,E2 -16579.527} C_VEL
LIN {X 0,Y 459.821,Z 437.841,A -85,B 0,C 180,E1 -16580.334,E2 -16580.334} C_VEL
LIN {X 0,Y 463.363,Z 378.031,A -85,B 0,C 180,E1 -16581.816,E2 -16581.816} C_VEL
LIN {X 0,Y 457.457,Z 366.213,A -85,B 0,C 180,E1 -16582.815,E2 -16582.815} C_VEL
LIN {X 0,Y 450.999,Z 355.314,A -85,B 0,C 180,E1 -16583.949,E2 -16583.949} C_VEL
LIN {X 0,Y 448.065,Z 350.873,A -85,B 0,C 180,E1 -16584.474,E2 -16584.474} C_VEL
LIN {X 0,Y 446.032,Z 347.409,A -85,B 0,C 180,E1 -16584.88,E2 -16584.88} C_VEL
LIN {X 0,Y 444.195,Z 345.076,A -85,B 0,C 180,E1 -16585.226,E2 -16585.226} C_VEL
LIN {X 0,Y 443.514,Z 342.801,A -85,B 0,C 180,E1 -16585.423,E2 -16585.423} C_VEL
LIN {X 0,Y 443.525,Z 342.798,A -85,B 0,C 180,E1 -16588.28,E2 -16588.28} C_VEL
LIN {X 0,Y 443.53,Z 342.795,A -85,B 0,C 180,E1 -16591.482,E2 -16591.482} C_VEL
LIN {X 0,Y 443.541,Z 342.789,A -85,B 0,C 180,E1 -16594.795,E2 -16594.795} C_VEL
LIN {X 0,Y 443.494,Z 342.792,A -85,B 0,C 180,E1 -16598.021,E2 -16598.021} C_VEL
LIN {X 0,Y 443.486,Z 342.795,A -85,B 0,C 180,E1 -16601.556,E2 -16601.556} C_VEL
LIN {X 0,Y 443.494,Z 342.795,A -85,B 0,C 180,E1 -16604.706,E2 -16604.706} C_VEL
LIN {X 0,Y 443.498,Z 342.795,A -85,B 0,C 180,E1 -16607.928,E2 -16607.928} C_VEL
LIN {X 0,Y 443.481,Z 342.803,A -85,B 0,C 180,E1 -16610.819,E2 -16610.819} C_VEL
LIN {X 0,Y 443.432,Z 342.81,A -85,B 0,C 180,E1 -16614.235,E2 -16614.235} C_VEL
LIN {X 0,Y 443.489,Z 342.924,A -85,B 0,C 180,E1 -16616.135,E2 -16616.135} C_VEL
LIN {X 0,Y 447.138,Z 357.145,A -85,B 0,C 180,E1 -16618.644,E2 -16618.644} C_VEL
LIN {X 0,Y 450.448,Z 372.325,A -85,B 0,C 180,E1 -16621.18,E2 -16621.18} C_VEL
LIN {X 0,Y 450.905,Z 375.718,A -85,B 0,C 180,E1 -16621.719,E2 -16621.719} C_VEL
LIN {X 0,Y 449.066,Z 394.571,A -85,B 0,C 180,E1 -16624.415,E2 -16624.415} C_VEL
LIN {X 0,Y 452.69,Z 416.894,A -85,B 0,C 180,E1 -16625.591,E2 -16625.591} C_VEL
LIN {X 0,Y 455.234,Z 435.26,A -85,B 0,C 180,E1 -16626.442,E2 -16626.442} C_VEL
LIN {X 0,Y 456.95,Z 451.366,A -85,B 0,C 180,E1 -16627.111,E2 -16627.111} C_VEL
LIN {X 0,Y 458.319,Z 475.31,A -85,B 0,C 180,E1 -16627.949,E2 -16627.949} C_VEL
LIN {X 0,Y 454.054,Z 554.803,A -85,B 0,C 180,E1 -16629.896,E2 -16629.896} C_VEL
LIN {X 0,Y 452.731,Z 570.488,A -85,B 0,C 180,E1 -16630.453,E2 -16630.453} C_VEL
LIN {X 0,Y 451.223,Z 583.768,A -85,B 0,C 180,E1 -16631.092,E2 -16631.092} C_VEL
LIN {X 0,Y 449.575,Z 599.372,A -85,B 0,C 180,E1 -16631.975,E2 -16631.975} C_VEL
LIN {X 0,Y 448.179,Z 611.46,A -85,B 0,C 180,E1 -16632.843,E2 -16632.843} C_VEL
LIN {X 0,Y 446.841,Z 622.777,A -85,B 0,C 180,E1 -16633.845,E2 -16633.845} C_VEL
LIN {X 0,Y 445.455,Z 633.208,A -85,B 0,C 180,E1 -16634.962,E2 -16634.962} C_VEL
LIN {X 0,Y 444.21,Z 643.647,A -85,B 0,C 180,E1 -16636.318,E2 -16636.318} C_VEL
LIN {X 0,Y 443.514,Z 651.092,A -85,B 0,C 180,E1 -16637.458,E2 -16637.458} C_VEL
LIN {X 0,Y 442.891,Z 661.852,A -85,B 0,C 180,E1 -16638.68,E2 -16638.68} C_VEL
LIN {X 0,Y 442.43,Z 671.297,A -85,B 0,C 180,E1 -16639.971,E2 -16639.971} C_VEL
LIN {X 0,Y 442.055,Z 679.642,A -85,B 0,C 180,E1 -16641.342,E2 -16641.342} C_VEL
LIN {X 0,Y 441.78,Z 687.6,A -85,B 0,C 180,E1 -16642.942,E2 -16642.942} C_VEL
LIN {X 0,Y 441.638,Z 693.886,A -85,B 0,C 180,E1 -16644.539,E2 -16644.539} C_VEL
LIN {X 0,Y 441.512,Z 698.114,A -85,B 0,C 180,E1 -16645.906,E2 -16645.906} C_VEL
LIN {X 0,Y 441.492,Z 701.358,A -85,B 0,C 180,E1 -16647.272,E2 -16647.272} C_VEL
LIN {X 0,Y 441.512,Z 704.326,A -85,B 0,C 180,E1 -16649.091,E2 -16649.091} C_VEL
LIN {X 0,Y 441.463,Z 705.783,A -85,B 0,C 180,E1 -16650.909,E2 -16650.909} C_VEL
LIN {X 0,Y 441.502,Z 705.944,A -85,B 0,C 180,E1 -16651.818,E2 -16651.818} C_VEL
LIN {X 0,Y 441.554,Z 705.141,A -85,B 0,C 180,E1 -16653.638,E2 -16653.638} C_VEL
LIN {X 0,Y 441.77,Z 702.878,A -85,B 0,C 180,E1 -16655.459,E2 -16655.459} C_VEL
LIN {X 0,Y 442.223,Z 699.106,A -85,B 0,C 180,E1 -16657.28,E2 -16657.28} C_VEL
LIN {X 0,Y 442.872,Z 693.761,A -85,B 0,C 180,E1 -16659.1,E2 -16659.1} C_VEL
LIN {X 0,Y 443.634,Z 688.548,A -85,B 0,C 180,E1 -16660.461,E2 -16660.461} C_VEL
LIN {X 0,Y 444.594,Z 682.249,A -85,B 0,C 180,E1 -16661.818,E2 -16661.818} C_VEL
LIN {X 0,Y 445.59,Z 674.99,A -85,B 0,C 180,E1 -16663.129,E2 -16663.129} C_VEL
LIN {X 0,Y 447,Z 665.657,A -85,B 0,C 180,E1 -16664.52,E2 -16664.52} C_VEL
LIN {X 0,Y 448.59,Z 654.809,A -85,B 0,C 180,E1 -16665.858,E2 -16665.858} C_VEL
LIN {X 0,Y 450.214,Z 642.675,A -85,B 0,C 180,E1 -16667.077,E2 -16667.077} C_VEL
LIN {X 0,Y 451.988,Z 629.13,A -85,B 0,C 180,E1 -16668.172,E2 -16668.172} C_VEL
LIN {X 0,Y 453.497,Z 615.696,A -85,B 0,C 180,E1 -16669.043,E2 -16669.043} C_VEL
LIN {X 0,Y 454.958,Z 600.498,A -85,B 0,C 180,E1 -16669.798,E2 -16669.798} C_VEL
LIN {X 0,Y 456.346,Z 584.571,A -85,B 0,C 180,E1 -16670.363,E2 -16670.363} C_VEL
LIN {X 0,Y 462.273,Z 486.885,A -85,B 0,C 180,E1 -16672.818,E2 -16672.818} C_VEL
LIN {X 0,Y 462.817,Z 475.21,A -85,B 0,C 180,E1 -16673.143,E2 -16673.143} C_VEL
LIN {X 0,Y 462.126,Z 459.124,A -85,B 0,C 180,E1 -16673.744,E2 -16673.744} C_VEL
LIN {X 0,Y 460.037,Z 437.959,A -85,B 0,C 180,E1 -16674.691,E2 -16674.691} C_VEL
LIN {X 0,Y 459.786,Z 427.748,A -85,B 0,C 180,E1 -16675.397,E2 -16675.397} C_VEL
LIN {X 0,Y 459.532,Z 409.783,A -85,B 0,C 180,E1 -16676.808,E2 -16676.808} C_VEL
LIN {X 0,Y 459.327,Z 395.564,A -85,B 0,C 180,E1 -16678.088,E2 -16678.088} C_VEL
LIN {X 0,Y 459.417,Z 385.597,A -85,B 0,C 180,E1 -16679.052,E2 -16679.052} C_VEL
LIN {X 0,Y 459.365,Z 380.278,A -85,B 0,C 180,E1 -16679.641,E2 -16679.641} C_VEL
LIN {X 0,Y 458.001,Z 370.607,A -85,B 0,C 180,E1 -16681.081,E2 -16681.081} C_VEL
LIN {X 0,Y 457.572,Z 366.981,A -85,B 0,C 180,E1 -16681.687,E2 -16681.687} C_VEL
LIN {X 0,Y 457.197,Z 365.806,A -85,B 0,C 180,E1 -16681.948,E2 -16681.948} C_VEL
LIN {X 0,Y 455.316,Z 362.431,A -85,B 0,C 180,E1 -16682.976,E2 -16682.976} C_VEL
LIN {X 0,Y 452.163,Z 357.313,A -85,B 0,C 180,E1 -16684.971,E2 -16684.971} C_VEL
LIN {X 0,Y 450.562,Z 355.107,A -85,B 0,C 180,E1 -16686.21,E2 -16686.21} C_VEL
LIN {X 0,Y 449.601,Z 352.977,A -85,B 0,C 180,E1 -16687.415,E2 -16687.415} C_VEL
LIN {X 0,Y 447.85,Z 351.05,A -85,B 0,C 180,E1 -16689.971,E2 -16689.971} C_VEL
LIN {X 0,Y 447.516,Z 350.651,A -85,B 0,C 180,E1 -16692.301,E2 -16692.301} C_VEL
LIN {X 0,Y 448.323,Z 351.666,A -85,B 0,C 180,E1 -16694.673,E2 -16694.673} C_VEL
LIN {X 0,Y 449.109,Z 352.665,A -85,B 0,C 180,E1 -16695.843,E2 -16695.843} C_VEL
LIN {X 0,Y 451.197,Z 357.332,A -85,B 0,C 180,E1 -16698.634,E2 -16698.634} C_VEL
LIN {X 0,Y 453.3,Z 362.154,A -85,B 0,C 180,E1 -16700.689,E2 -16700.689} C_VEL
LIN {X 0,Y 456.105,Z 368.976,A -85,B 0,C 180,E1 -16702.994,E2 -16702.994} C_VEL
LIN {X 0,Y 458.985,Z 377.297,A -85,B 0,C 180,E1 -16705.242,E2 -16705.242} C_VEL
LIN {X 0,Y 461.36,Z 386.284,A -85,B 0,C 180,E1 -16707.264,E2 -16707.264} C_VEL
LIN {X 0,Y 463.231,Z 395.472,A -85,B 0,C 180,E1 -16709.062,E2 -16709.062} C_VEL
LIN {X 0,Y 463.315,Z 398.207,A -85,B 0,C 180,E1 -16709.512,E2 -16709.512} C_VEL
LIN {X 0,Y 460.037,Z 421.148,A -85,B 0,C 180,E1 -16712.579,E2 -16712.579} C_VEL
LIN {X 0,Y 457.689,Z 440.108,A -85,B 0,C 180,E1 -16715.035,E2 -16715.035} C_VEL
LIN {X 0,Y 460.927,Z 457.208,A -85,B 0,C 180,E1 -16715.978,E2 -16715.978} C_VEL
LIN {X 0,Y 463.157,Z 473.555,A -85,B 0,C 180,E1 -16716.743,E2 -16716.743} C_VEL
LIN {X 0,Y 463.252,Z 477.503,A -85,B 0,C 180,E1 -16716.879,E2 -16716.879} C_VEL
LIN {X 0,Y 458.101,Z 561.894,A -85,B 0,C 180,E1 -16718.982,E2 -16718.982} C_VEL
LIN {X 0,Y 456.747,Z 584.055,A -85,B 0,C 180,E1 -16719.549,E2 -16719.549} C_VEL
LIN {X 0,Y 455.516,Z 598.212,A -85,B 0,C 180,E1 -16720.075,E2 -16720.075} C_VEL
LIN {X 0,Y 453.918,Z 613.806,A -85,B 0,C 180,E1 -16720.858,E2 -16720.858} C_VEL
LIN {X 0,Y 452.442,Z 627.062,A -85,B 0,C 180,E1 -16721.73,E2 -16721.73} C_VEL
LIN {X 0,Y 450.664,Z 640.449,A -85,B 0,C 180,E1 -16722.824,E2 -16722.824} C_VEL
LIN {X 0,Y 448.994,Z 652.565,A -85,B 0,C 180,E1 -16724.041,E2 -16724.041} C_VEL
LIN {X 0,Y 447.52,Z 662.596,A -85,B 0,C 180,E1 -16725.266,E2 -16725.266} C_VEL
LIN {X 0,Y 445.997,Z 672.227,A -85,B 0,C 180,E1 -16726.683,E2 -16726.683} C_VEL
LIN {X 0,Y 444.883,Z 680.56,A -85,B 0,C 180,E1 -16728.19,E2 -16728.19} C_VEL
LIN {X 0,Y 443.833,Z 686.797,A -85,B 0,C 180,E1 -16729.544,E2 -16729.544} C_VEL
LIN {X 0,Y 443.049,Z 691.961,A -85,B 0,C 180,E1 -16730.904,E2 -16730.904} C_VEL
LIN {X 0,Y 442.284,Z 697.26,A -85,B 0,C 180,E1 -16732.722,E2 -16732.722} C_VEL
LIN {X 0,Y 441.762,Z 700.995,A -85,B 0,C 180,E1 -16734.541,E2 -16734.541} C_VEL
LIN {X 0,Y 441.521,Z 703.242,A -85,B 0,C 180,E1 -16736.362,E2 -16736.362} C_VEL
LIN {X 0,Y 441.422,Z 704.046,A -85,B 0,C 180,E1 -16738.182,E2 -16738.182} C_VEL
LIN {X 0,Y 441.409,Z 703.377,A -85,B 0,C 180,E1 -16740,E2 -16740} C_VEL
LIN {X 0,Y 441.422,Z 701.209,A -85,B 0,C 180,E1 -16741.819,E2 -16741.819} C_VEL
LIN {X 0,Y 441.457,Z 697.526,A -85,B 0,C 180,E1 -16743.639,E2 -16743.639} C_VEL
LIN {X 0,Y 441.551,Z 693.704,A -85,B 0,C 180,E1 -16745.006,E2 -16745.006} C_VEL
LIN {X 0,Y 441.694,Z 688.887,A -85,B 0,C 180,E1 -16746.374,E2 -16746.374} C_VEL
LIN {X 0,Y 441.939,Z 681.818,A -85,B 0,C 180,E1 -16747.972,E2 -16747.972} C_VEL
LIN {X 0,Y 442.426,Z 673.025,A -85,B 0,C 180,E1 -16749.569,E2 -16749.569} C_VEL
LIN {X 0,Y 442.895,Z 663.815,A -85,B 0,C 180,E1 -16750.94,E2 -16750.94} C_VEL
LIN {X 0,Y 443.56,Z 652.681,A -85,B 0,C 180,E1 -16752.309,E2 -16752.309} C_VEL
LIN {X 0,Y 444.157,Z 641.356,A -85,B 0,C 180,E1 -16753.451,E2 -16753.451} C_VEL
LIN {X 0,Y 444.9,Z 629.038,A -85,B 0,C 180,E1 -16754.474,E2 -16754.474} C_VEL
LIN {X 0,Y 445.713,Z 615.556,A -85,B 0,C 180,E1 -16755.379,E2 -16755.379} C_VEL
LIN {X 0,Y 446.197,Z 602.713,A -85,B 0,C 180,E1 -16756.062,E2 -16756.062} C_VEL
LIN {X 0,Y 446.785,Z 588.288,A -85,B 0,C 180,E1 -16756.642,E2 -16756.642} C_VEL
LIN {X 0,Y 447.299,Z 572.635,A -85,B 0,C 180,E1 -16757.069,E2 -16757.069} C_VEL
LIN {X 0,Y 449.757,Z 469.875,A -85,B 0,C 180,E1 -16759.273,E2 -16759.273} C_VEL
LIN {X 0,Y 446.79,Z 439.497,A -85,B 0,C 180,E1 -16760.051,E2 -16760.051} C_VEL
LIN {X 0,Y 448.391,Z 411.554,A -85,B 0,C 180,E1 -16763.475,E2 -16763.475} C_VEL
LIN {X 0,Y 449.908,Z 386.192,A -85,B 0,C 180,E1 -16766.59,E2 -16766.59} C_VEL
LIN {X 0,Y 450.563,Z 374.361,A -85,B 0,C 180,E1 -16768.052,E2 -16768.052} C_VEL
LIN {X 0,Y 446.771,Z 356.822,A -85,B 0,C 180,E1 -16770.426,E2 -16770.426} C_VEL
LIN {X 0,Y 443.58,Z 342.788,A -85,B 0,C 180,E1 -16772.365,E2 -16772.365} C_VEL
LIN {X 0,Y 443.532,Z 342.793,A -85,B 0,C 180,E1 -16775.755,E2 -16775.755} C_VEL
LIN {X 0,Y 443.518,Z 342.797,A -85,B 0,C 180,E1 -16779.299,E2 -16779.299} C_VEL
LIN {X 0,Y 443.515,Z 342.796,A -85,B 0,C 180,E1 -16782.774,E2 -16782.774} C_VEL
LIN {X 0,Y 443.522,Z 342.791,A -85,B 0,C 180,E1 -16785.982,E2 -16785.982} C_VEL
LIN {X 0,Y 443.517,Z 342.794,A -85,B 0,C 180,E1 -16789.294,E2 -16789.294} C_VEL
LIN {X 0,Y 443.499,Z 342.796,A -85,B 0,C 180,E1 -16792.156,E2 -16792.156} C_VEL
LIN {X 0,Y 443.53,Z 342.791,A -85,B 0,C 180,E1 -16795.352,E2 -16795.352} C_VEL
LIN {X 0,Y 443.539,Z 342.795,A -85,B 0,C 180,E1 -16798.591,E2 -16798.591} C_VEL
LIN {X 0,Y 443.526,Z 342.791,A -85,B 0,C 180,E1 -16801.72,E2 -16801.72} C_VEL
LIN {X 0,Y 443.491,Z 342.798,A -85,B 0,C 180,E1 -16804.759,E2 -16804.759} C_VEL
LIN {X 0,Y 443.514,Z 342.794,A -85,B 0,C 180,E1 -16807.726,E2 -16807.726} C_VEL
LIN {X 0,Y 443.563,Z 342.79,A -85,B 0,C 180,E1 -16810.633,E2 -16810.633} C_VEL
LIN {X 0,Y 443.576,Z 342.792,A -85,B 0,C 180,E1 -16814.17,E2 -16814.17} C_VEL
LIN {X 0,Y 443.565,Z 342.793,A -85,B 0,C 180,E1 -16814.282,E2 -16814.282} C_VEL
LIN {X 0,Y 452.252,Z 365.857,A -85,B 0,C 180,E1 -16815.064,E2 -16815.064} C_VEL
LIN {X 0,Y 451.213,Z 456.482,A -85,B 0,C 180,E1 -16816.508,E2 -16816.508} C_VEL
LIN {X 0,Y 451.103,Z 470.903,A -85,B 0,C 180,E1 -16816.846,E2 -16816.846} C_VEL
LIN {X 0,Y 450.774,Z 484.145,A -85,B 0,C 180,E1 -16817.321,E2 -16817.321} C_VEL
LIN {X 0,Y 450.157,Z 497.721,A -85,B 0,C 180,E1 -16817.988,E2 -16817.988} C_VEL
LIN {X 0,Y 449.469,Z 509.951,A -85,B 0,C 180,E1 -16818.767,E2 -16818.767} C_VEL
LIN {X 0,Y 448.771,Z 522.312,A -85,B 0,C 180,E1 -16819.759,E2 -16819.759} C_VEL
LIN {X 0,Y 447.809,Z 533.816,A -85,B 0,C 180,E1 -16820.888,E2 -16820.888} C_VEL
LIN {X 0,Y 446.856,Z 544.091,A -85,B 0,C 180,E1 -16822.117,E2 -16822.117} C_VEL
LIN {X 0,Y 445.833,Z 553.393,A -85,B 0,C 180,E1 -16823.46,E2 -16823.46} C_VEL
LIN {X 0,Y 444.966,Z 562.255,A -85,B 0,C 180,E1 -16825.033,E2 -16825.033} C_VEL
LIN {X 0,Y 444.283,Z 568.497,A -85,B 0,C 180,E1 -16826.384,E2 -16826.384} C_VEL
LIN {X 0,Y 443.786,Z 573.633,A -85,B 0,C 180,E1 -16827.739,E2 -16827.739} C_VEL
LIN {X 0,Y 443.278,Z 579.065,A -85,B 0,C 180,E1 -16829.547,E2 -16829.547} C_VEL
LIN {X 0,Y 443.063,Z 582.106,A -85,B 0,C 180,E1 -16830.906,E2 -16830.906} C_VEL
LIN {X 0,Y 442.992,Z 584.955,A -85,B 0,C 180,E1 -16832.719,E2 -16832.719} C_VEL
LIN {X 0,Y 442.858,Z 586.509,A -85,B 0,C 180,E1 -16834.536,E2 -16834.536} C_VEL
LIN {X 0,Y 443.027,Z 586.753,A -85,B 0,C 180,E1 -16836.354,E2 -16836.354} C_VEL
LIN {X 0,Y 443.252,Z 585.716,A -85,B 0,C 180,E1 -16838.177,E2 -16838.177} C_VEL
LIN {X 0,Y 443.604,Z 583.365,A -85,B 0,C 180,E1 -16840.003,E2 -16840.003} C_VEL
LIN {X 0,Y 444.372,Z 579.589,A -85,B 0,C 180,E1 -16841.825,E2 -16841.825} C_VEL
LIN {X 0,Y 445.176,Z 574.212,A -85,B 0,C 180,E1 -16843.666,E2 -16843.666} C_VEL
LIN {X 0,Y 444.93,Z 571.888,A -85,B 0,C 180,E1 -16844.361,E2 -16844.361} C_VEL
LIN {X 0,Y 442.811,Z 567.901,A -85,B 0,C 180,E1 -16845.502,E2 -16845.502} C_VEL
LIN {X 0,Y 440.737,Z 563.464,A -85,B 0,C 180,E1 -16846.621,E2 -16846.621} C_VEL
LIN {X 0,Y 440.565,Z 560.276,A -85,B 0,C 180,E1 -16847.273,E2 -16847.273} C_VEL
LIN {X 0,Y 441.812,Z 551.653,A -85,B 0,C 180,E1 -16848.726,E2 -16848.726} C_VEL
LIN {X 0,Y 443.161,Z 541.667,A -85,B 0,C 180,E1 -16850.107,E2 -16850.107} C_VEL
LIN {X 0,Y 444.484,Z 530.468,A -85,B 0,C 180,E1 -16851.368,E2 -16851.368} C_VEL
LIN {X 0,Y 445.633,Z 519.21,A -85,B 0,C 180,E1 -16852.406,E2 -16852.406} C_VEL
LIN {X 0,Y 446.765,Z 506.896,A -85,B 0,C 180,E1 -16853.321,E2 -16853.321} C_VEL
LIN {X 0,Y 447.478,Z 493.326,A -85,B 0,C 180,E1 -16854.126,E2 -16854.126} C_VEL
LIN {X 0,Y 448.132,Z 479.493,A -85,B 0,C 180,E1 -16854.732,E2 -16854.732} C_VEL
LIN {X 0,Y 448.43,Z 465.617,A -85,B 0,C 180,E1 -16855.16,E2 -16855.16} C_VEL
LIN {X 0,Y 448.852,Z 437.019,A -85,B 0,C 180,E1 -16855.661,E2 -16855.661} C_VEL
LIN {X 0,Y 450.058,Z 374.072,A -85,B 0,C 180,E1 -16856.671,E2 -16856.671} C_VEL
LIN {X 0,Y 439.817,Z 351.356,A -85,B 0,C 180,E1 -16857.68,E2 -16857.68} C_VEL
LIN {X 0,Y 436.57,Z 344.299,A -85,B 0,C 180,E1 -16858.009,E2 -16858.009} C_VEL
LIN {X 0,Y 436.455,Z 343.674,A -85,B 0,C 180,E1 -16858.033,E2 -16858.033} C_VEL
LIN {X 0,Y 436.419,Z 343.68,A -85,B 0,C 180,E1 -16860.904,E2 -16860.904} C_VEL
LIN {X 0,Y 436.389,Z 343.685,A -85,B 0,C 180,E1 -16864.18,E2 -16864.18} C_VEL
LIN {X 0,Y 436.432,Z 343.679,A -85,B 0,C 180,E1 -16867.581,E2 -16867.581} C_VEL
LIN {X 0,Y 436.421,Z 343.681,A -85,B 0,C 180,E1 -16871.032,E2 -16871.032} C_VEL
LIN {X 0,Y 436.437,Z 343.682,A -85,B 0,C 180,E1 -16873.762,E2 -16873.762} C_VEL
LIN {X 0,Y 436.452,Z 343.678,A -85,B 0,C 180,E1 -16876.362,E2 -16876.362} C_VEL
LIN {X 0,Y 436.425,Z 343.676,A -85,B 0,C 180,E1 -16878.967,E2 -16878.967} C_VEL
LIN {X 0,Y 436.428,Z 343.65,A -85,B 0,C 180,E1 -16882.419,E2 -16882.419} C_VEL
LIN {X 0,Y 436.427,Z 343.669,A -85,B 0,C 180,E1 -16885.824,E2 -16885.824} C_VEL
LIN {X 0,Y 436.427,Z 343.67,A -85,B 0,C 180,E1 -16889.097,E2 -16889.097} C_VEL
LIN {X 0,Y 436.468,Z 343.671,A -85,B 0,C 180,E1 -16892.264,E2 -16892.264} C_VEL
LIN {X 0,Y 436.444,Z 343.671,A -85,B 0,C 180,E1 -16895.337,E2 -16895.337} C_VEL
LIN {X 0,Y 436.458,Z 343.665,A -85,B 0,C 180,E1 -16898.562,E2 -16898.562} C_VEL
LIN {X 0,Y 436.522,Z 343.664,A -85,B 0,C 180,E1 -16899.545,E2 -16899.545} C_VEL
LIN {X 0,Y 442.359,Z 364.219,A -85,B 0,C 180,E1 -16900.188,E2 -16900.188} C_VEL
LIN {X 0,Y 440.329,Z 461.781,A -85,B 0,C 180,E1 -16902.318,E2 -16902.318} C_VEL
LIN {X 0,Y 440.129,Z 477.008,A -85,B 0,C 180,E1 -16902.84,E2 -16902.84} C_VEL
LIN {X 0,Y 439.638,Z 491.341,A -85,B 0,C 180,E1 -16903.513,E2 -16903.513} C_VEL
LIN {X 0,Y 439.101,Z 505.49,A -85,B 0,C 180,E1 -16904.384,E2 -16904.384} C_VEL
LIN {X 0,Y 438.518,Z 519.001,A -85,B 0,C 180,E1 -16905.429,E2 -16905.429} C_VEL
LIN {X 0,Y 437.844,Z 531.221,A -85,B 0,C 180,E1 -16906.587,E2 -16906.587} C_VEL
LIN {X 0,Y 437.469,Z 541.493,A -85,B 0,C 180,E1 -16907.767,E2 -16907.767} C_VEL
LIN {X 0,Y 436.93,Z 551.515,A -85,B 0,C 180,E1 -16909.142,E2 -16909.142} C_VEL
LIN {X 0,Y 436.372,Z 561.247,A -85,B 0,C 180,E1 -16910.763,E2 -16910.763} C_VEL
LIN {X 0,Y 436.054,Z 568.061,A -85,B 0,C 180,E1 -16912.152,E2 -16912.152} C_VEL
LIN {X 0,Y 435.858,Z 573.698,A -85,B 0,C 180,E1 -16913.541,E2 -16913.541} C_VEL
LIN {X 0,Y 435.72,Z 579.517,A -85,B 0,C 180,E1 -16915.339,E2 -16915.339} C_VEL
LIN {X 0,Y 435.755,Z 581.969,A -85,B 0,C 180,E1 -16916.313,E2 -16916.313} C_VEL
LIN {X 0,Y 435.775,Z 585.466,A -85,B 0,C 180,E1 -16918.158,E2 -16918.158} C_VEL
LIN {X 0,Y 435.897,Z 587.512,A -85,B 0,C 180,E1 -16920,E2 -16920} C_VEL
LIN {X 0,Y 436.288,Z 588.12,A -85,B 0,C 180,E1 -16921.84,E2 -16921.84} C_VEL
LIN {X 0,Y 436.89,Z 587.235,A -85,B 0,C 180,E1 -16923.677,E2 -16923.677} C_VEL
LIN {X 0,Y 437.738,Z 584.9,A -85,B 0,C 180,E1 -16925.509,E2 -16925.509} C_VEL
LIN {X 0,Y 438.639,Z 581.109,A -85,B 0,C 180,E1 -16927.339,E2 -16927.339} C_VEL
LIN {X 0,Y 439.577,Z 577.554,A -85,B 0,C 180,E1 -16928.573,E2 -16928.573} C_VEL
LIN {X 0,Y 440.827,Z 572.186,A -85,B 0,C 180,E1 -16930.066,E2 -16930.066} C_VEL
LIN {X 0,Y 442.176,Z 565.048,A -85,B 0,C 180,E1 -16931.652,E2 -16931.652} C_VEL
LIN {X 0,Y 443.582,Z 557.51,A -85,B 0,C 180,E1 -16933.004,E2 -16933.004} C_VEL
LIN {X 0,Y 445.061,Z 548.477,A -85,B 0,C 180,E1 -16934.352,E2 -16934.352} C_VEL
LIN {X 0,Y 446.364,Z 539.459,A -85,B 0,C 180,E1 -16935.472,E2 -16935.472} C_VEL
LIN {X 0,Y 448.022,Z 527.498,A -85,B 0,C 180,E1 -16936.695,E2 -16936.695} C_VEL
LIN {X 0,Y 449.605,Z 514.298,A -85,B 0,C 180,E1 -16937.78,E2 -16937.78} C_VEL
LIN {X 0,Y 450.856,Z 500.707,A -85,B 0,C 180,E1 -16938.676,E2 -16938.676} C_VEL
LIN {X 0,Y 451.695,Z 487.685,A -85,B 0,C 180,E1 -16939.357,E2 -16939.357} C_VEL
LIN {X 0,Y 452.441,Z 473.404,A -85,B 0,C 180,E1 -16939.913,E2 -16939.913} C_VEL
LIN {X 0,Y 453.179,Z 453.314,A -85,B 0,C 180,E1 -16940.469,E2 -16940.469} C_VEL
